LIN {X -75.070,Y -30.211,Z -61.011,A -90.000,B 90.000,C 0.000} C_DIS
LIN {X -75.157,Y -30.255,Z -61.208,A -90.000,B 90.000,C 0.000} C_DIS
LIN {X -75.236,Y -30.297,Z -61.411,A -90.000,B 90.000,C 0.000} C_DIS
LIN {X -75.317,Y -30.342,Z -61.633,A -90.000,B 90.000,C 0.000} C_DIS
LIN {X -75.352,Y -30.355,Z -61.731,A -90.000,B 90.000,C 0.000} C_DIS
LIN {X -75.467,Y -30.405,Z -62.109,A -90.000,B 90.000,C 0.000} C_DIS
LIN {X -75.521,Y -30.436,Z -62.301,A -90.000,B 90.000,C 0.000} C_DIS
LIN {X -75.551,Y -30.454,Z -62.421,A -90.000,B 90.000,C 0.000} C_DIS
LIN {X -75.584,Y -30.470,Z -62.557,A -90.000,B 90.000,C 0.000} C_DIS
LIN {X -75.622,Y -30.482,Z -62.719,A -90.000,B 90.000,C 0.000} C_DIS
LIN {X -75.673,Y -30.490,Z -62.969,A -90.000,B 90.000,C 0.000} C_DIS
LIN {X -75.693,Y -30.495,Z -63.078,A -90.000,B 90.000,C 0.000} C_DIS
LIN {X -75.763,Y -30.514,Z -63.484,A -90.000,B 90.000,C 0.000} C_DIS
LIN {X -75.780,Y -30.517,Z -63.601,A -90.000,B 90.000,C 0.000} C_DIS
LIN {X -75.801,Y -30.514,Z -63.775,A -90.000,B 90.000,C 0.000} C_DIS
LIN {X -75.817,Y -30.506,Z -63.923,A -90.000,B 90.000,C 0.000} C_DIS
LIN {X -75.841,Y -30.490,Z -64.222,A -90.000,B 90.000,C 0.000} C_DIS
LIN {X -75.855,Y -30.471,Z -64.525,A -90.000,B 90.000,C 0.000} C_DIS
LIN {X -75.859,Y -30.448,Z -64.759,A -90.000,B 90.000,C 0.000} C_DIS
LIN {X -75.857,Y -30.400,Z -65.089,A -90.000,B 90.000,C 0.000} C_DIS
LIN {X -75.852,Y -30.383,Z -65.199,A -90.000,B 90.000,C 0.000} C_DIS
LIN {X -75.840,Y -30.342,Z -65.434,A -90.000,B 90.000,C 0.000} C_DIS
LIN {X -75.824,Y -30.298,Z -65.657,A -90.000,B 90.000,C 0.000} C_DIS
LIN {X -75.790,Y -30.221,Z -66.013,A -90.000,B 90.000,C 0.000} C_DIS
LIN {X -75.781,Y -30.202,Z -66.095,A -90.000,B 90.000,C 0.000} C_DIS
LIN {X -75.717,Y -30.104,Z -66.510,A -90.000,B 90.000,C 0.000} C_DIS
LIN {X -75.684,Y -30.057,Z -66.702,A -90.000,B 90.000,C 0.000} C_DIS
LIN {X -75.646,Y -30.005,Z -66.902,A -90.000,B 90.000,C 0.000} C_DIS
LIN {X -75.556,Y -29.899,Z -67.292,A -90.000,B 90.000,C 0.000} C_DIS
LIN {X -75.456,Y -29.777,Z -67.697,A -90.000,B 90.000,C 0.000} C_DIS
LIN {X -75.421,Y -29.737,Z -67.825,A -90.000,B 90.000,C 0.000} C_DIS
LIN {X -75.365,Y -29.676,Z -68.020,A -90.000,B 90.000,C 0.000} C_DIS
LIN {X -75.295,Y -29.600,Z -68.251,A -90.000,B 90.000,C 0.000} C_DIS
LIN {X -75.175,Y -29.475,Z -68.600,A -90.000,B 90.000,C 0.000} C_DIS
LIN {X -75.139,Y -29.441,Z -68.694,A -90.000,B 90.000,C 0.000} C_DIS
LIN {X -75.103,Y -29.407,Z -68.780,A -90.000,B 90.000,C 0.000} C_DIS
LIN {X -75.036,Y -29.353,Z -68.939,A -90.000,B 90.000,C 0.000} C_DIS
LIN {X -74.986,Y -29.308,Z -69.055,A -90.000,B 90.000,C 0.000} C_DIS
LIN {X -74.986,Y -60.000,Z -69.055,A -90.000,B 90.000,C 0.000} C_DIS
LIN {X -75.487,Y -60.000,Z -57.775,A -90.000,B 90.000,C 0.000} C_DIS
LIN {X -75.487,Y -29.308,Z -57.775,A -90.000,B 90.000,C 0.000} C_DIS
LIN {X -75.588,Y -29.374,Z -57.912,A -90.000,B 90.000,C 0.000} C_DIS
LIN {X -75.705,Y -29.444,Z -58.076,A -90.000,B 90.000,C 0.000} C_DIS
LIN {X -75.899,Y -29.577,Z -58.363,A -90.000,B 90.000,C 0.000} C_DIS
LIN {X -76.016,Y -29.661,Z -58.548,A -90.000,B 90.000,C 0.000} C_DIS
LIN {X -76.226,Y -29.805,Z -58.898,A -90.000,B 90.000,C 0.000} C_DIS
LIN {X -76.268,Y -29.838,Z -58.968,A -90.000,B 90.000,C 0.000} C_DIS
LIN {X -76.317,Y -29.873,Z -59.050,A -90.000,B 90.000,C 0.000} C_DIS
LIN {X -76.378,Y -29.912,Z -59.154,A -90.000,B 90.000,C 0.000} C_DIS
LIN {X -76.468,Y -29.969,Z -59.312,A -90.000,B 90.000,C 0.000} C_DIS
LIN {X -76.540,Y -30.015,Z -59.446,A -90.000,B 90.000,C 0.000} C_DIS
LIN {X -76.686,Y -30.114,Z -59.738,A -90.000,B 90.000,C 0.000} C_DIS
LIN {X -76.865,Y -30.240,Z -60.127,A -90.000,B 90.000,C 0.000} C_DIS
LIN {X -76.997,Y -30.336,Z -60.429,A -90.000,B 90.000,C 0.000} C_DIS
LIN {X -77.105,Y -30.422,Z -60.708,A -90.000,B 90.000,C 0.000} C_DIS
LIN {X -77.183,Y -30.483,Z -60.928,A -90.000,B 90.000,C 0.000} C_DIS
LIN {X -77.250,Y -30.536,Z -61.129,A -90.000,B 90.000,C 0.000} C_DIS
LIN {X -77.333,Y -30.609,Z -61.412,A -90.000,B 90.000,C 0.000} C_DIS
LIN {X -77.363,Y -30.633,Z -61.516,A -90.000,B 90.000,C 0.000} C_DIS
LIN {X -77.423,Y -30.670,Z -61.730,A -90.000,B 90.000,C 0.000} C_DIS
LIN {X -77.467,Y -30.699,Z -61.904,A -90.000,B 90.000,C 0.000} C_DIS
LIN {X -77.546,Y -30.756,Z -62.248,A -90.000,B 90.000,C 0.000} C_DIS
LIN {X -77.612,Y -30.808,Z -62.596,A -90.000,B 90.000,C 0.000} C_DIS
LIN {X -77.629,Y -30.818,Z -62.691,A -90.000,B 90.000,C 0.000} C_DIS
LIN {X -77.639,Y -30.821,Z -62.751,A -90.000,B 90.000,C 0.000} C_DIS
LIN {X -77.695,Y -30.830,Z -63.070,A -90.000,B 90.000,C 0.000} C_DIS
LIN {X -77.728,Y -30.839,Z -63.278,A -90.000,B 90.000,C 0.000} C_DIS
LIN {X -77.744,Y -30.843,Z -63.408,A -90.000,B 90.000,C 0.000} C_DIS
LIN {X -77.759,Y -30.844,Z -63.540,A -90.000,B 90.000,C 0.000} C_DIS
LIN {X -77.780,Y -30.841,Z -63.734,A -90.000,B 90.000,C 0.000} C_DIS
LIN {X -77.808,Y -30.822,Z -64.070,A -90.000,B 90.000,C 0.000} C_DIS
LIN {X -77.823,Y -30.805,Z -64.362,A -90.000,B 90.000,C 0.000} C_DIS
LIN {X -77.830,Y -30.789,Z -64.526,A -90.000,B 90.000,C 0.000} C_DIS
LIN {X -77.835,Y -30.757,Z -64.759,A -90.000,B 90.000,C 0.000} C_DIS
LIN {X -77.834,Y -30.725,Z -64.999,A -90.000,B 90.000,C 0.000} C_DIS
LIN {X -77.832,Y -30.689,Z -65.212,A -90.000,B 90.000,C 0.000} C_DIS
LIN {X -77.815,Y -30.623,Z -65.585,A -90.000,B 90.000,C 0.000} C_DIS
LIN {X -77.791,Y -30.565,Z -65.906,A -90.000,B 90.000,C 0.000} C_DIS
LIN {X -77.756,Y -30.496,Z -66.260,A -90.000,B 90.000,C 0.000} C_DIS
LIN {X -77.732,Y -30.456,Z -66.455,A -90.000,B 90.000,C 0.000} C_DIS
LIN {X -77.659,Y -30.352,Z -66.915,A -90.000,B 90.000,C 0.000} C_DIS
LIN {X -77.634,Y -30.314,Z -67.066,A -90.000,B 90.000,C 0.000} C_DIS
LIN {X -77.579,Y -30.237,Z -67.357,A -90.000,B 90.000,C 0.000} C_DIS
LIN {X -77.481,Y -30.105,Z -67.792,A -90.000,B 90.000,C 0.000} C_DIS
LIN {X -77.383,Y -29.974,Z -68.194,A -90.000,B 90.000,C 0.000} C_DIS
LIN {X -77.376,Y -29.962,Z -68.225,A -90.000,B 90.000,C 0.000} C_DIS
LIN {X -77.320,Y -29.872,Z -68.440,A -90.000,B 90.000,C 0.000} C_DIS
LIN {X -77.199,Y -29.695,Z -68.857,A -90.000,B 90.000,C 0.000} C_DIS
LIN {X -77.135,Y -29.612,Z -69.048,A -90.000,B 90.000,C 0.000} C_DIS
LIN {X -77.071,Y -29.520,Z -69.234,A -90.000,B 90.000,C 0.000} C_DIS
LIN {X -77.025,Y -29.457,Z -69.361,A -90.000,B 90.000,C 0.000} C_DIS
LIN {X -76.963,Y -29.379,Z -69.514,A -90.000,B 90.000,C 0.000} C_DIS
LIN {X -76.909,Y -29.308,Z -69.641,A -90.000,B 90.000,C 0.000} C_DIS
LIN {X -76.877,Y -29.271,Z -69.720,A -90.000,B 90.000,C 0.000} C_DIS
LIN {X -76.826,Y -29.187,Z -69.873,A -90.000,B 90.000,C 0.000} C_DIS
LIN {X -76.806,Y -29.148,Z -69.945,A -90.000,B 90.000,C 0.000} C_DIS
LIN {X -76.778,Y -29.074,Z -70.083,A -90.000,B 90.000,C 0.000} C_DIS
LIN {X -76.770,Y -29.039,Z -70.149,A -90.000,B 90.000,C 0.000} C_DIS
LIN {X -76.764,Y -28.972,Z -70.272,A -90.000,B 90.000,C 0.000} C_DIS
LIN {X -76.772,Y -28.913,Z -70.387,A -90.000,B 90.000,C 0.000} C_DIS
LIN {X -76.792,Y -28.861,Z -70.491,A -90.000,B 90.000,C 0.000} C_DIS
LIN {X -76.824,Y -28.814,Z -70.586,A -90.000,B 90.000,C 0.000} C_DIS
LIN {X -76.844,Y -28.794,Z -70.630,A -90.000,B 90.000,C 0.000} C_DIS
LIN {X -76.892,Y -28.757,Z -70.710,A -90.000,B 90.000,C 0.000} C_DIS
LIN {X -76.950,Y -28.723,Z -70.781,A -90.000,B 90.000,C 0.000} C_DIS
LIN {X -77.017,Y -28.694,Z -70.841,A -90.000,B 90.000,C 0.000} C_DIS
LIN {X -77.054,Y -28.682,Z -70.868,A -90.000,B 90.000,C 0.000} C_DIS
LIN {X -77.132,Y -28.662,Z -70.913,A -90.000,B 90.000,C 0.000} C_DIS
LIN {X -77.218,Y -28.647,Z -70.948,A -90.000,B 90.000,C 0.000} C_DIS
LIN {X -77.310,Y -28.637,Z -70.973,A -90.000,B 90.000,C 0.000} C_DIS
LIN {X -77.406,Y -28.632,Z -70.988,A -90.000,B 90.000,C 0.000} C_DIS
LIN {X -77.456,Y -28.631,Z -70.992,A -90.000,B 90.000,C 0.000} C_DIS
LIN {X -77.559,Y -28.634,Z -70.991,A -90.000,B 90.000,C 0.000} C_DIS
LIN {X -77.612,Y -28.637,Z -70.987,A -90.000,B 90.000,C 0.000} C_DIS
LIN {X -77.719,Y -28.649,Z -70.970,A -90.000,B 90.000,C 0.000} C_DIS
LIN {X -77.774,Y -28.657,Z -70.958,A -90.000,B 90.000,C 0.000} C_DIS
LIN {X -77.884,Y -28.677,Z -70.926,A -90.000,B 90.000,C 0.000} C_DIS
LIN {X -77.994,Y -28.703,Z -70.883,A -90.000,B 90.000,C 0.000} C_DIS
LIN {X -78.104,Y -28.734,Z -70.830,A -90.000,B 90.000,C 0.000} C_DIS
LIN {X -78.159,Y -28.751,Z -70.799,A -90.000,B 90.000,C 0.000} C_DIS
LIN {X -78.267,Y -28.789,Z -70.729,A -90.000,B 90.000,C 0.000} C_DIS
LIN {X -78.373,Y -28.832,Z -70.649,A -90.000,B 90.000,C 0.000} C_DIS
LIN {X -78.425,Y -28.856,Z -70.604,A -90.000,B 90.000,C 0.000} C_DIS
LIN {X -78.525,Y -28.906,Z -70.507,A -90.000,B 90.000,C 0.000} C_DIS
LIN {X -78.622,Y -28.962,Z -70.399,A -90.000,B 90.000,C 0.000} C_DIS
LIN {X -78.713,Y -29.024,Z -70.280,A -90.000,B 90.000,C 0.000} C_DIS
LIN {X -78.798,Y -29.092,Z -70.149,A -90.000,B 90.000,C 0.000} C_DIS
LIN {X -78.877,Y -29.163,Z -70.008,A -90.000,B 90.000,C 0.000} C_DIS
LIN {X -78.947,Y -29.236,Z -69.855,A -90.000,B 90.000,C 0.000} C_DIS
LIN {X -78.979,Y -29.275,Z -69.774,A -90.000,B 90.000,C 0.000} C_DIS
LIN {X -79.009,Y -29.308,Z -69.690,A -90.000,B 90.000,C 0.000} C_DIS
LIN {X -79.097,Y -29.432,Z -69.431,A -90.000,B 90.000,C 0.000} C_DIS
LIN {X -79.136,Y -29.488,Z -69.310,A -90.000,B 90.000,C 0.000} C_DIS
LIN {X -79.250,Y -29.666,Z -68.921,A -90.000,B 90.000,C 0.000} C_DIS
LIN {X -79.335,Y -29.794,Z -68.596,A -90.000,B 90.000,C 0.000} C_DIS
LIN {X -79.365,Y -29.841,Z -68.472,A -90.000,B 90.000,C 0.000} C_DIS
LIN {X -79.464,Y -29.983,Z -68.059,A -90.000,B 90.000,C 0.000} C_DIS
LIN {X -79.538,Y -30.078,Z -67.731,A -90.000,B 90.000,C 0.000} C_DIS
LIN {X -79.614,Y -30.175,Z -67.319,A -90.000,B 90.000,C 0.000} C_DIS
LIN {X -79.633,Y -30.199,Z -67.204,A -90.000,B 90.000,C 0.000} C_DIS
LIN {X -79.716,Y -30.304,Z -66.656,A -90.000,B 90.000,C 0.000} C_DIS
LIN {X -79.743,Y -30.346,Z -66.432,A -90.000,B 90.000,C 0.000} C_DIS
LIN {X -79.782,Y -30.423,Z -66.029,A -90.000,B 90.000,C 0.000} C_DIS
LIN {X -79.809,Y -30.494,Z -65.654,A -90.000,B 90.000,C 0.000} C_DIS
LIN {X -79.829,Y -30.583,Z -65.203,A -90.000,B 90.000,C 0.000} C_DIS
LIN {X -79.832,Y -30.637,Z -64.931,A -90.000,B 90.000,C 0.000} C_DIS
LIN {X -79.831,Y -30.688,Z -64.643,A -90.000,B 90.000,C 0.000} C_DIS
LIN {X -79.826,Y -30.718,Z -64.432,A -90.000,B 90.000,C 0.000} C_DIS
LIN {X -79.812,Y -30.760,Z -64.109,A -90.000,B 90.000,C 0.000} C_DIS
LIN {X -79.800,Y -30.786,Z -63.901,A -90.000,B 90.000,C 0.000} C_DIS
LIN {X -79.776,Y -30.821,Z -63.606,A -90.000,B 90.000,C 0.000} C_DIS
LIN {X -79.748,Y -30.833,Z -63.329,A -90.000,B 90.000,C 0.000} C_DIS
LIN {X -79.709,Y -30.846,Z -63.005,A -90.000,B 90.000,C 0.000} C_DIS
LIN {X -79.682,Y -30.850,Z -62.829,A -90.000,B 90.000,C 0.000} C_DIS
LIN {X -79.652,Y -30.849,Z -62.653,A -90.000,B 90.000,C 0.000} C_DIS
LIN {X -79.597,Y -30.835,Z -62.339,A -90.000,B 90.000,C 0.000} C_DIS
LIN {X -79.527,Y -30.809,Z -61.960,A -90.000,B 90.000,C 0.000} C_DIS
LIN {X -79.497,Y -30.797,Z -61.808,A -90.000,B 90.000,C 0.000} C_DIS
LIN {X -79.476,Y -30.786,Z -61.720,A -90.000,B 90.000,C 0.000} C_DIS
LIN {X -79.404,Y -30.737,Z -61.408,A -90.000,B 90.000,C 0.000} C_DIS
LIN {X -79.348,Y -30.703,Z -61.187,A -90.000,B 90.000,C 0.000} C_DIS
LIN {X -79.256,Y -30.648,Z -60.864,A -90.000,B 90.000,C 0.000} C_DIS
LIN {X -79.165,Y -30.590,Z -60.555,A -90.000,B 90.000,C 0.000} C_DIS
LIN {X -79.089,Y -30.544,Z -60.326,A -90.000,B 90.000,C 0.000} C_DIS
LIN {X -79.019,Y -30.504,Z -60.123,A -90.000,B 90.000,C 0.000} C_DIS
LIN {X -78.959,Y -30.470,Z -59.961,A -90.000,B 90.000,C 0.000} C_DIS
LIN {X -78.853,Y -30.411,Z -59.686,A -90.000,B 90.000,C 0.000} C_DIS
LIN {X -78.755,Y -30.359,Z -59.461,A -90.000,B 90.000,C 0.000} C_DIS
LIN {X -78.672,Y -30.312,Z -59.273,A -90.000,B 90.000,C 0.000} C_DIS
LIN {X -78.596,Y -30.271,Z -59.110,A -90.000,B 90.000,C 0.000} C_DIS
LIN {X -78.494,Y -30.219,Z -58.891,A -90.000,B 90.000,C 0.000} C_DIS
LIN {X -78.326,Y -30.122,Z -58.553,A -90.000,B 90.000,C 0.000} C_DIS
LIN {X -78.288,Y -30.099,Z -58.479,A -90.000,B 90.000,C 0.000} C_DIS
LIN {X -78.218,Y -30.055,Z -58.347,A -90.000,B 90.000,C 0.000} C_DIS
LIN {X -78.075,Y -29.971,Z -58.098,A -90.000,B 90.000,C 0.000} C_DIS
LIN {X -77.857,Y -29.832,Z -57.731,A -90.000,B 90.000,C 0.000} C_DIS
LIN {X -77.697,Y -29.704,Z -57.464,A -90.000,B 90.000,C 0.000} C_DIS
LIN {X -77.595,Y -29.626,Z -57.303,A -90.000,B 90.000,C 0.000} C_DIS
LIN {X -77.526,Y -29.571,Z -57.198,A -90.000,B 90.000,C 0.000} C_DIS
LIN {X -77.371,Y -29.450,Z -56.969,A -90.000,B 90.000,C 0.000} C_DIS
LIN {X -77.219,Y -29.308,Z -56.755,A -90.000,B 90.000,C 0.000} C_DIS
LIN {X -77.219,Y -60.000,Z -56.755,A -90.000,B 90.000,C 0.000} C_DIS
LIN {X -81.350,Y -60.000,Z -68.141,A -90.000,B 90.000,C 0.000} C_DIS
LIN {X -81.350,Y -29.308,Z -68.141,A -90.000,B 90.000,C 0.000} C_DIS
LIN {X -81.402,Y -29.373,Z -67.896,A -90.000,B 90.000,C 0.000} C_DIS
LIN {X -81.465,Y -29.458,Z -67.573,A -90.000,B 90.000,C 0.000} C_DIS
LIN {X -81.521,Y -29.531,Z -67.237,A -90.000,B 90.000,C 0.000} C_DIS
LIN {X -81.592,Y -29.618,Z -66.755,A -90.000,B 90.000,C 0.000} C_DIS
LIN {X -81.618,Y -29.659,Z -66.531,A -90.000,B 90.000,C 0.000} C_DIS
LIN {X -81.648,Y -29.714,Z -66.217,A -90.000,B 90.000,C 0.000} C_DIS
LIN {X -81.663,Y -29.743,Z -66.039,A -90.000,B 90.000,C 0.000} C_DIS
LIN {X -81.678,Y -29.782,Z -65.813,A -90.000,B 90.000,C 0.000} C_DIS
LIN {X -81.694,Y -29.828,Z -65.576,A -90.000,B 90.000,C 0.000} C_DIS
LIN {X -81.701,Y -29.857,Z -65.445,A -90.000,B 90.000,C 0.000} C_DIS
LIN {X -81.721,Y -29.943,Z -65.094,A -90.000,B 90.000,C 0.000} C_DIS
LIN {X -81.731,Y -30.038,Z -64.718,A -90.000,B 90.000,C 0.000} C_DIS
LIN {X -81.733,Y -30.072,Z -64.570,A -90.000,B 90.000,C 0.000} C_DIS
LIN {X -81.733,Y -30.147,Z -64.227,A -90.000,B 90.000,C 0.000} C_DIS
LIN {X -81.724,Y -30.226,Z -63.852,A -90.000,B 90.000,C 0.000} C_DIS
LIN {X -81.716,Y -30.257,Z -63.679,A -90.000,B 90.000,C 0.000} C_DIS
LIN {X -81.701,Y -30.298,Z -63.446,A -90.000,B 90.000,C 0.000} C_DIS
LIN {X -81.674,Y -30.339,Z -63.114,A -90.000,B 90.000,C 0.000} C_DIS
LIN {X -81.627,Y -30.371,Z -62.693,A -90.000,B 90.000,C 0.000} C_DIS
LIN {X -81.593,Y -30.390,Z -62.458,A -90.000,B 90.000,C 0.000} C_DIS
LIN {X -81.549,Y -30.402,Z -62.175,A -90.000,B 90.000,C 0.000} C_DIS
LIN {X -81.528,Y -30.406,Z -62.039,A -90.000,B 90.000,C 0.000} C_DIS
LIN {X -81.477,Y -30.401,Z -61.750,A -90.000,B 90.000,C 0.000} C_DIS
LIN {X -81.442,Y -30.392,Z -61.558,A -90.000,B 90.000,C 0.000} C_DIS
LIN {X -81.416,Y -30.389,Z -61.420,A -90.000,B 90.000,C 0.000} C_DIS
LIN {X -81.399,Y -30.384,Z -61.342,A -90.000,B 90.000,C 0.000} C_DIS
LIN {X -81.384,Y -30.383,Z -61.267,A -90.000,B 90.000,C 0.000} C_DIS
LIN {X -81.312,Y -30.366,Z -60.936,A -90.000,B 90.000,C 0.000} C_DIS
LIN {X -81.256,Y -30.355,Z -60.699,A -90.000,B 90.000,C 0.000} C_DIS
LIN {X -81.162,Y -30.339,Z -60.343,A -90.000,B 90.000,C 0.000} C_DIS
LIN {X -81.080,Y -30.321,Z -60.045,A -90.000,B 90.000,C 0.000} C_DIS
LIN {X -81.050,Y -30.312,Z -59.943,A -90.000,B 90.000,C 0.000} C_DIS
LIN {X -80.964,Y -30.301,Z -59.670,A -90.000,B 90.000,C 0.000} C_DIS
LIN {X -80.864,Y -30.289,Z -59.375,A -90.000,B 90.000,C 0.000} C_DIS
LIN {X -80.828,Y -30.288,Z -59.273,A -90.000,B 90.000,C 0.000} C_DIS
LIN {X -80.786,Y -30.286,Z -59.158,A -90.000,B 90.000,C 0.000} C_DIS
LIN {X -80.714,Y -30.275,Z -58.969,A -90.000,B 90.000,C 0.000} C_DIS
LIN {X -80.639,Y -30.260,Z -58.789,A -90.000,B 90.000,C 0.000} C_DIS
LIN {X -80.544,Y -30.249,Z -58.566,A -90.000,B 90.000,C 0.000} C_DIS
LIN {X -80.414,Y -30.228,Z -58.278,A -90.000,B 90.000,C 0.000} C_DIS
LIN {X -80.309,Y -30.205,Z -58.051,A -90.000,B 90.000,C 0.000} C_DIS
LIN {X -80.245,Y -30.189,Z -57.919,A -90.000,B 90.000,C 0.000} C_DIS
LIN {X -80.160,Y -30.161,Z -57.749,A -90.000,B 90.000,C 0.000} C_DIS
LIN {X -80.048,Y -30.115,Z -57.527,A -90.000,B 90.000,C 0.000} C_DIS
LIN {X -79.993,Y -30.094,Z -57.426,A -90.000,B 90.000,C 0.000} C_DIS
LIN {X -79.803,Y -30.021,Z -57.093,A -90.000,B 90.000,C 0.000} C_DIS
LIN {X -79.744,Y -29.999,Z -56.993,A -90.000,B 90.000,C 0.000} C_DIS
LIN {X -79.506,Y -29.860,Z -56.595,A -90.000,B 90.000,C 0.000} C_DIS
LIN {X -79.371,Y -29.767,Z -56.373,A -90.000,B 90.000,C 0.000} C_DIS
LIN {X -79.307,Y -29.724,Z -56.272,A -90.000,B 90.000,C 0.000} C_DIS
LIN {X -79.170,Y -29.618,Z -56.060,A -90.000,B 90.000,C 0.000} C_DIS
LIN {X -79.030,Y -29.514,Z -55.855,A -90.000,B 90.000,C 0.000} C_DIS
LIN {X -78.810,Y -29.308,Z -55.544,A -90.000,B 90.000,C 0.000} C_DIS
LIN {X -78.614,Y -29.120,Z -55.273,A -90.000,B 90.000,C 0.000} C_DIS
LIN {X -78.524,Y -29.030,Z -55.153,A -90.000,B 90.000,C 0.000} C_DIS
LIN {X -78.438,Y -28.942,Z -55.043,A -90.000,B 90.000,C 0.000} C_DIS
LIN {X -78.357,Y -28.857,Z -54.942,A -90.000,B 90.000,C 0.000} C_DIS
LIN {X -78.281,Y -28.774,Z -54.851,A -90.000,B 90.000,C 0.000} C_DIS
LIN {X -78.210,Y -28.693,Z -54.769,A -90.000,B 90.000,C 0.000} C_DIS
LIN {X -78.143,Y -28.615,Z -54.696,A -90.000,B 90.000,C 0.000} C_DIS
LIN {X -78.081,Y -28.539,Z -54.633,A -90.000,B 90.000,C 0.000} C_DIS
LIN {X -77.970,Y -28.403,Z -54.532,A -90.000,B 90.000,C 0.000} C_DIS
LIN {X -77.921,Y -28.357,Z -54.494,A -90.000,B 90.000,C 0.000} C_DIS
LIN {X -77.876,Y -28.317,Z -54.465,A -90.000,B 90.000,C 0.000} C_DIS
LIN {X -77.835,Y -28.283,Z -54.444,A -90.000,B 90.000,C 0.000} C_DIS
LIN {X -77.782,Y -28.246,Z -54.427,A -90.000,B 90.000,C 0.000} C_DIS
LIN {X -77.752,Y -28.230,Z -54.426,A -90.000,B 90.000,C 0.000} C_DIS
LIN {X -77.738,Y -28.225,Z -54.428,A -90.000,B 90.000,C 0.000} C_DIS
LIN {X -77.714,Y -28.220,Z -54.438,A -90.000,B 90.000,C 0.000} C_DIS
LIN {X -77.693,Y -28.223,Z -54.455,A -90.000,B 90.000,C 0.000} C_DIS
LIN {X -77.684,Y -28.227,Z -54.467,A -90.000,B 90.000,C 0.000} C_DIS
LIN {X -77.670,Y -28.241,Z -54.495,A -90.000,B 90.000,C 0.000} C_DIS
LIN {X -77.658,Y -28.261,Z -54.530,A -90.000,B 90.000,C 0.000} C_DIS
LIN {X -77.648,Y -28.303,Z -54.595,A -90.000,B 90.000,C 0.000} C_DIS
LIN {X -77.646,Y -28.337,Z -54.646,A -90.000,B 90.000,C 0.000} C_DIS
LIN {X -77.652,Y -28.421,Z -54.768,A -90.000,B 90.000,C 0.000} C_DIS
LIN {X -77.660,Y -28.469,Z -54.838,A -90.000,B 90.000,C 0.000} C_DIS
LIN {X -77.685,Y -28.577,Z -54.995,A -90.000,B 90.000,C 0.000} C_DIS
LIN {X -77.747,Y -28.769,Z -55.271,A -90.000,B 90.000,C 0.000} C_DIS
LIN {X -77.802,Y -28.916,Z -55.480,A -90.000,B 90.000,C 0.000} C_DIS
LIN {X -77.834,Y -28.990,Z -55.592,A -90.000,B 90.000,C 0.000} C_DIS
LIN {X -77.906,Y -29.137,Z -55.829,A -90.000,B 90.000,C 0.000} C_DIS
LIN {X -77.946,Y -29.208,Z -55.953,A -90.000,B 90.000,C 0.000} C_DIS
LIN {X -77.988,Y -29.278,Z -56.082,A -90.000,B 90.000,C 0.000} C_DIS
LIN {X -78.033,Y -29.346,Z -56.214,A -90.000,B 90.000,C 0.000} C_DIS
LIN {X -78.080,Y -29.411,Z -56.350,A -90.000,B 90.000,C 0.000} C_DIS
LIN {X -78.129,Y -29.486,Z -56.490,A -90.000,B 90.000,C 0.000} C_DIS
LIN {X -78.235,Y -29.629,Z -56.778,A -90.000,B 90.000,C 0.000} C_DIS
LIN {X -78.348,Y -29.756,Z -57.079,A -90.000,B 90.000,C 0.000} C_DIS
LIN {X -78.470,Y -29.868,Z -57.390,A -90.000,B 90.000,C 0.000} C_DIS
LIN {X -78.598,Y -29.981,Z -57.710,A -90.000,B 90.000,C 0.000} C_DIS
LIN {X -78.734,Y -30.079,Z -58.037,A -90.000,B 90.000,C 0.000} C_DIS
LIN {X -78.875,Y -30.163,Z -58.371,A -90.000,B 90.000,C 0.000} C_DIS
LIN {X -79.022,Y -30.244,Z -58.711,A -90.000,B 90.000,C 0.000} C_DIS
LIN {X -79.174,Y -30.317,Z -59.053,A -90.000,B 90.000,C 0.000} C_DIS
LIN {X -79.330,Y -30.377,Z -59.399,A -90.000,B 90.000,C 0.000} C_DIS
LIN {X -79.490,Y -30.440,Z -59.745,A -90.000,B 90.000,C 0.000} C_DIS
LIN {X -79.654,Y -30.500,Z -60.091,A -90.000,B 90.000,C 0.000} C_DIS
LIN {X -79.820,Y -30.551,Z -60.435,A -90.000,B 90.000,C 0.000} C_DIS
LIN {X -79.989,Y -30.596,Z -60.776,A -90.000,B 90.000,C 0.000} C_DIS
LIN {X -80.159,Y -30.632,Z -61.113,A -90.000,B 90.000,C 0.000} C_DIS
LIN {X -80.331,Y -30.651,Z -61.443,A -90.000,B 90.000,C 0.000} C_DIS
LIN {X -80.503,Y -30.664,Z -61.767,A -90.000,B 90.000,C 0.000} C_DIS
LIN {X -80.589,Y -30.663,Z -61.926,A -90.000,B 90.000,C 0.000} C_DIS
LIN {X -80.675,Y -30.656,Z -62.083,A -90.000,B 90.000,C 0.000} C_DIS
LIN {X -80.761,Y -30.642,Z -62.237,A -90.000,B 90.000,C 0.000} C_DIS
LIN {X -81.018,Y -30.587,Z -62.683,A -90.000,B 90.000,C 0.000} C_DIS
LIN {X -81.103,Y -30.565,Z -62.826,A -90.000,B 90.000,C 0.000} C_DIS
LIN {X -81.187,Y -30.537,Z -62.965,A -90.000,B 90.000,C 0.000} C_DIS
LIN {X -81.271,Y -30.504,Z -63.101,A -90.000,B 90.000,C 0.000} C_DIS
LIN {X -81.354,Y -30.465,Z -63.233,A -90.000,B 90.000,C 0.000} C_DIS
LIN {X -81.437,Y -30.420,Z -63.362,A -90.000,B 90.000,C 0.000} C_DIS
LIN {X -81.518,Y -30.372,Z -63.486,A -90.000,B 90.000,C 0.000} C_DIS
LIN {X -81.599,Y -30.322,Z -63.606,A -90.000,B 90.000,C 0.000} C_DIS
LIN {X -81.680,Y -30.269,Z -63.722,A -90.000,B 90.000,C 0.000} C_DIS
LIN {X -81.759,Y -30.215,Z -63.834,A -90.000,B 90.000,C 0.000} C_DIS
LIN {X -81.914,Y -30.104,Z -64.043,A -90.000,B 90.000,C 0.000} C_DIS
LIN {X -81.990,Y -30.047,Z -64.140,A -90.000,B 90.000,C 0.000} C_DIS
LIN {X -82.064,Y -29.988,Z -64.232,A -90.000,B 90.000,C 0.000} C_DIS
LIN {X -82.138,Y -29.927,Z -64.319,A -90.000,B 90.000,C 0.000} C_DIS
LIN {X -82.210,Y -29.866,Z -64.400,A -90.000,B 90.000,C 0.000} C_DIS
LIN {X -82.281,Y -29.804,Z -64.476,A -90.000,B 90.000,C 0.000} C_DIS
LIN {X -82.350,Y -29.742,Z -64.545,A -90.000,B 90.000,C 0.000} C_DIS
LIN {X -82.417,Y -29.680,Z -64.609,A -90.000,B 90.000,C 0.000} C_DIS
LIN {X -82.483,Y -29.618,Z -64.667,A -90.000,B 90.000,C 0.000} C_DIS
LIN {X -82.547,Y -29.557,Z -64.718,A -90.000,B 90.000,C 0.000} C_DIS
LIN {X -82.640,Y -29.468,Z -64.783,A -90.000,B 90.000,C 0.000} C_DIS
LIN {X -82.729,Y -29.381,Z -64.832,A -90.000,B 90.000,C 0.000} C_DIS
LIN {X -82.813,Y -29.299,Z -64.866,A -90.000,B 90.000,C 0.000} C_DIS
LIN {X -82.893,Y -29.225,Z -64.883,A -90.000,B 90.000,C 0.000} C_DIS
LIN {X -82.968,Y -29.161,Z -64.884,A -90.000,B 90.000,C 0.000} C_DIS
LIN {X -83.015,Y -29.125,Z -64.874,A -90.000,B 90.000,C 0.000} C_DIS
LIN {X -83.037,Y -29.108,Z -64.867,A -90.000,B 90.000,C 0.000} C_DIS
LIN {X -83.081,Y -29.079,Z -64.845,A -90.000,B 90.000,C 0.000} C_DIS
LIN {X -83.122,Y -29.055,Z -64.816,A -90.000,B 90.000,C 0.000} C_DIS
LIN {X -83.141,Y -29.044,Z -64.798,A -90.000,B 90.000,C 0.000} C_DIS
LIN {X -83.178,Y -29.027,Z -64.756,A -90.000,B 90.000,C 0.000} C_DIS
LIN {X -83.213,Y -29.015,Z -64.705,A -90.000,B 90.000,C 0.000} C_DIS
LIN {X -83.245,Y -29.008,Z -64.646,A -90.000,B 90.000,C 0.000} C_DIS
LIN {X -83.274,Y -29.008,Z -64.578,A -90.000,B 90.000,C 0.000} C_DIS
LIN {X -83.300,Y -29.013,Z -64.500,A -90.000,B 90.000,C 0.000} C_DIS
LIN {X -83.323,Y -29.023,Z -64.413,A -90.000,B 90.000,C 0.000} C_DIS
LIN {X -83.344,Y -29.037,Z -64.317,A -90.000,B 90.000,C 0.000} C_DIS
LIN {X -83.361,Y -29.053,Z -64.211,A -90.000,B 90.000,C 0.000} C_DIS
LIN {X -83.375,Y -29.075,Z -64.096,A -90.000,B 90.000,C 0.000} C_DIS
LIN {X -83.390,Y -29.117,Z -63.903,A -90.000,B 90.000,C 0.000} C_DIS
LIN {X -83.396,Y -29.151,Z -63.763,A -90.000,B 90.000,C 0.000} C_DIS
LIN {X -83.399,Y -29.184,Z -63.611,A -90.000,B 90.000,C 0.000} C_DIS
LIN {X -83.399,Y -29.215,Z -63.450,A -90.000,B 90.000,C 0.000} C_DIS
LIN {X -83.387,Y -29.280,Z -63.094,A -90.000,B 90.000,C 0.000} C_DIS
LIN {X -83.375,Y -29.308,Z -62.899,A -90.000,B 90.000,C 0.000} C_DIS
LIN {X -83.340,Y -29.392,Z -62.367,A -90.000,B 90.000,C 0.000} C_DIS
LIN {X -83.321,Y -29.434,Z -62.141,A -90.000,B 90.000,C 0.000} C_DIS
LIN {X -83.293,Y -29.471,Z -61.871,A -90.000,B 90.000,C 0.000} C_DIS
LIN {X -83.279,Y -29.487,Z -61.740,A -90.000,B 90.000,C 0.000} C_DIS
LIN {X -83.251,Y -29.525,Z -61.458,A -90.000,B 90.000,C 0.000} C_DIS
LIN {X -83.233,Y -29.543,Z -61.294,A -90.000,B 90.000,C 0.000} C_DIS
LIN {X -83.206,Y -29.576,Z -61.053,A -90.000,B 90.000,C 0.000} C_DIS
LIN {X -83.177,Y -29.602,Z -60.844,A -90.000,B 90.000,C 0.000} C_DIS
LIN {X -83.140,Y -29.653,Z -60.548,A -90.000,B 90.000,C 0.000} C_DIS
LIN {X -83.085,Y -29.698,Z -60.228,A -90.000,B 90.000,C 0.000} C_DIS
LIN {X -83.039,Y -29.734,Z -59.992,A -90.000,B 90.000,C 0.000} C_DIS
LIN {X -83.018,Y -29.753,Z -59.880,A -90.000,B 90.000,C 0.000} C_DIS
LIN {X -82.978,Y -29.784,Z -59.689,A -90.000,B 90.000,C 0.000} C_DIS
LIN {X -82.952,Y -29.805,Z -59.564,A -90.000,B 90.000,C 0.000} C_DIS
LIN {X -82.909,Y -29.828,Z -59.388,A -90.000,B 90.000,C 0.000} C_DIS
LIN {X -82.831,Y -29.867,Z -59.101,A -90.000,B 90.000,C 0.000} C_DIS
LIN {X -82.800,Y -29.883,Z -58.994,A -90.000,B 90.000,C 0.000} C_DIS
LIN {X -82.745,Y -29.914,Z -58.807,A -90.000,B 90.000,C 0.000} C_DIS
LIN {X -82.687,Y -29.932,Z -58.625,A -90.000,B 90.000,C 0.000} C_DIS
LIN {X -82.667,Y -29.935,Z -58.567,A -90.000,B 90.000,C 0.000} C_DIS
LIN {X -82.629,Y -29.950,Z -58.459,A -90.000,B 90.000,C 0.000} C_DIS
LIN {X -82.569,Y -29.967,Z -58.287,A -90.000,B 90.000,C 0.000} C_DIS
LIN {X -82.465,Y -29.987,Z -58.020,A -90.000,B 90.000,C 0.000} C_DIS
LIN {X -82.412,Y -29.996,Z -57.890,A -90.000,B 90.000,C 0.000} C_DIS
LIN {X -82.280,Y -30.022,Z -57.579,A -90.000,B 90.000,C 0.000} C_DIS
LIN {X -82.107,Y -30.032,Z -57.192,A -90.000,B 90.000,C 0.000} C_DIS
LIN {X -81.997,Y -30.031,Z -56.962,A -90.000,B 90.000,C 0.000} C_DIS
LIN {X -81.911,Y -30.024,Z -56.787,A -90.000,B 90.000,C 0.000} C_DIS
LIN {X -81.809,Y -30.011,Z -56.586,A -90.000,B 90.000,C 0.000} C_DIS
LIN {X -81.720,Y -29.990,Z -56.422,A -90.000,B 90.000,C 0.000} C_DIS
LIN {X -81.578,Y -29.953,Z -56.170,A -90.000,B 90.000,C 0.000} C_DIS
LIN {X -81.449,Y -29.911,Z -55.951,A -90.000,B 90.000,C 0.000} C_DIS
LIN {X -81.328,Y -29.870,Z -55.746,A -90.000,B 90.000,C 0.000} C_DIS
LIN {X -81.274,Y -29.847,Z -55.655,A -90.000,B 90.000,C 0.000} C_DIS
LIN {X -81.057,Y -29.725,Z -55.297,A -90.000,B 90.000,C 0.000} C_DIS
LIN {X -81.027,Y -29.707,Z -55.250,A -90.000,B 90.000,C 0.000} C_DIS
LIN {X -80.840,Y -29.582,Z -54.961,A -90.000,B 90.000,C 0.000} C_DIS
LIN {X -80.659,Y -29.453,Z -54.695,A -90.000,B 90.000,C 0.000} C_DIS
LIN {X -80.550,Y -29.376,Z -54.540,A -90.000,B 90.000,C 0.000} C_DIS
LIN {X -80.478,Y -29.308,Z -54.439,A -90.000,B 90.000,C 0.000} C_DIS
LIN {X -80.342,Y -29.188,Z -54.248,A -90.000,B 90.000,C 0.000} C_DIS
LIN {X -80.223,Y -29.065,Z -54.084,A -90.000,B 90.000,C 0.000} C_DIS
LIN {X -80.032,Y -28.856,Z -53.832,A -90.000,B 90.000,C 0.000} C_DIS
LIN {X -79.960,Y -28.781,Z -53.742,A -90.000,B 90.000,C 0.000} C_DIS
LIN {X -79.879,Y -28.699,Z -53.651,A -90.000,B 90.000,C 0.000} C_DIS
LIN {X -79.843,Y -28.665,Z -53.617,A -90.000,B 90.000,C 0.000} C_DIS
LIN {X -79.830,Y -28.655,Z -53.608,A -90.000,B 90.000,C 0.000} C_DIS
LIN {X -79.820,Y -28.648,Z -53.604,A -90.000,B 90.000,C 0.000} C_DIS
LIN {X -79.814,Y -28.647,Z -53.605,A -90.000,B 90.000,C 0.000} C_DIS
LIN {X -79.810,Y -28.649,Z -53.611,A -90.000,B 90.000,C 0.000} C_DIS
LIN {X -79.810,Y -28.656,Z -53.622,A -90.000,B 90.000,C 0.000} C_DIS
LIN {X -79.819,Y -28.681,Z -53.657,A -90.000,B 90.000,C 0.000} C_DIS
LIN {X -79.871,Y -28.773,Z -53.780,A -90.000,B 90.000,C 0.000} C_DIS
LIN {X -79.966,Y -28.911,Z -53.966,A -90.000,B 90.000,C 0.000} C_DIS
LIN {X -80.100,Y -29.094,Z -54.208,A -90.000,B 90.000,C 0.000} C_DIS
LIN {X -80.181,Y -29.193,Z -54.348,A -90.000,B 90.000,C 0.000} C_DIS
LIN {X -80.270,Y -29.292,Z -54.500,A -90.000,B 90.000,C 0.000} C_DIS
LIN {X -80.366,Y -29.388,Z -54.662,A -90.000,B 90.000,C 0.000} C_DIS
LIN {X -80.470,Y -29.479,Z -54.834,A -90.000,B 90.000,C 0.000} C_DIS
LIN {X -80.580,Y -29.564,Z -55.015,A -90.000,B 90.000,C 0.000} C_DIS
LIN {X -80.819,Y -29.730,Z -55.399,A -90.000,B 90.000,C 0.000} C_DIS
LIN {X -80.947,Y -29.806,Z -55.601,A -90.000,B 90.000,C 0.000} C_DIS
LIN {X -81.080,Y -29.871,Z -55.808,A -90.000,B 90.000,C 0.000} C_DIS
LIN {X -81.216,Y -29.924,Z -56.020,A -90.000,B 90.000,C 0.000} C_DIS
LIN {X -81.357,Y -29.963,Z -56.234,A -90.000,B 90.000,C 0.000} C_DIS
LIN {X -81.501,Y -29.996,Z -56.452,A -90.000,B 90.000,C 0.000} C_DIS
LIN {X -81.648,Y -30.026,Z -56.671,A -90.000,B 90.000,C 0.000} C_DIS
LIN {X -81.797,Y -30.043,Z -56.891,A -90.000,B 90.000,C 0.000} C_DIS
LIN {X -81.947,Y -30.046,Z -57.110,A -90.000,B 90.000,C 0.000} C_DIS
LIN {X -82.252,Y -30.026,Z -57.546,A -90.000,B 90.000,C 0.000} C_DIS
LIN {X -82.405,Y -30.002,Z -57.760,A -90.000,B 90.000,C 0.000} C_DIS
LIN {X -82.558,Y -29.976,Z -57.971,A -90.000,B 90.000,C 0.000} C_DIS
LIN {X -82.710,Y -29.944,Z -58.176,A -90.000,B 90.000,C 0.000} C_DIS
LIN {X -83.011,Y -29.858,Z -58.571,A -90.000,B 90.000,C 0.000} C_DIS
LIN {X -83.158,Y -29.805,Z -58.758,A -90.000,B 90.000,C 0.000} C_DIS
LIN {X -83.302,Y -29.748,Z -58.937,A -90.000,B 90.000,C 0.000} C_DIS
LIN {X -83.443,Y -29.691,Z -59.106,A -90.000,B 90.000,C 0.000} C_DIS
LIN {X -83.581,Y -29.625,Z -59.266,A -90.000,B 90.000,C 0.000} C_DIS
LIN {X -83.714,Y -29.558,Z -59.415,A -90.000,B 90.000,C 0.000} C_DIS
LIN {X -83.843,Y -29.493,Z -59.553,A -90.000,B 90.000,C 0.000} C_DIS
LIN {X -83.967,Y -29.425,Z -59.678,A -90.000,B 90.000,C 0.000} C_DIS
LIN {X -84.026,Y -29.390,Z -59.735,A -90.000,B 90.000,C 0.000} C_DIS
LIN {X -84.196,Y -29.288,Z -59.886,A -90.000,B 90.000,C 0.000} C_DIS
LIN {X -84.301,Y -29.227,Z -59.968,A -90.000,B 90.000,C 0.000} C_DIS
LIN {X -84.399,Y -29.170,Z -60.034,A -90.000,B 90.000,C 0.000} C_DIS
LIN {X -84.445,Y -29.142,Z -60.060,A -90.000,B 90.000,C 0.000} C_DIS
LIN {X -84.531,Y -29.092,Z -60.100,A -90.000,B 90.000,C 0.000} C_DIS
LIN {X -84.571,Y -29.070,Z -60.113,A -90.000,B 90.000,C 0.000} C_DIS
LIN {X -84.609,Y -29.050,Z -60.122,A -90.000,B 90.000,C 0.000} C_DIS
LIN {X -84.644,Y -29.032,Z -60.125,A -90.000,B 90.000,C 0.000} C_DIS
LIN {X -84.693,Y -29.010,Z -60.122,A -90.000,B 90.000,C 0.000} C_DIS
LIN {X -84.723,Y -28.999,Z -60.113,A -90.000,B 90.000,C 0.000} C_DIS
LIN {X -84.763,Y -28.988,Z -60.090,A -90.000,B 90.000,C 0.000} C_DIS
LIN {X -84.787,Y -28.984,Z -60.068,A -90.000,B 90.000,C 0.000} C_DIS
LIN {X -84.817,Y -28.983,Z -60.024,A -90.000,B 90.000,C 0.000} C_DIS
LIN {X -84.834,Y -28.987,Z -59.988,A -90.000,B 90.000,C 0.000} C_DIS
LIN {X -84.854,Y -28.998,Z -59.924,A -90.000,B 90.000,C 0.000} C_DIS
LIN {X -84.864,Y -29.009,Z -59.873,A -90.000,B 90.000,C 0.000} C_DIS
LIN {X -84.875,Y -29.040,Z -59.754,A -90.000,B 90.000,C 0.000} C_DIS
LIN {X -84.874,Y -29.080,Z -59.609,A -90.000,B 90.000,C 0.000} C_DIS
LIN {X -84.860,Y -29.128,Z -59.439,A -90.000,B 90.000,C 0.000} C_DIS
LIN {X -84.833,Y -29.182,Z -59.242,A -90.000,B 90.000,C 0.000} C_DIS
LIN {X -84.792,Y -29.246,Z -59.018,A -90.000,B 90.000,C 0.000} C_DIS
LIN {X -84.767,Y -29.281,Z -58.895,A -90.000,B 90.000,C 0.000} C_DIS
LIN {X -84.738,Y -29.308,Z -58.764,A -90.000,B 90.000,C 0.000} C_DIS
LIN {X -84.700,Y -29.353,Z -58.602,A -90.000,B 90.000,C 0.000} C_DIS
LIN {X -84.641,Y -29.410,Z -58.370,A -90.000,B 90.000,C 0.000} C_DIS
LIN {X -84.614,Y -29.435,Z -58.271,A -90.000,B 90.000,C 0.000} C_DIS
LIN {X -84.542,Y -29.484,Z -58.027,A -90.000,B 90.000,C 0.000} C_DIS
LIN {X -84.492,Y -29.517,Z -57.865,A -90.000,B 90.000,C 0.000} C_DIS
LIN {X -84.412,Y -29.565,Z -57.622,A -90.000,B 90.000,C 0.000} C_DIS
LIN {X -84.377,Y -29.588,Z -57.520,A -90.000,B 90.000,C 0.000} C_DIS
LIN {X -84.248,Y -29.648,Z -57.176,A -90.000,B 90.000,C 0.000} C_DIS
LIN {X -84.198,Y -29.670,Z -57.049,A -90.000,B 90.000,C 0.000} C_DIS
LIN {X -84.050,Y -29.714,Z -56.695,A -90.000,B 90.000,C 0.000} C_DIS
LIN {X -83.892,Y -29.751,Z -56.334,A -90.000,B 90.000,C 0.000} C_DIS
LIN {X -83.785,Y -29.772,Z -56.104,A -90.000,B 90.000,C 0.000} C_DIS
LIN {X -83.688,Y -29.788,Z -55.901,A -90.000,B 90.000,C 0.000} C_DIS
LIN {X -83.607,Y -29.794,Z -55.737,A -90.000,B 90.000,C 0.000} C_DIS
LIN {X -83.523,Y -29.792,Z -55.574,A -90.000,B 90.000,C 0.000} C_DIS
LIN {X -83.447,Y -29.786,Z -55.433,A -90.000,B 90.000,C 0.000} C_DIS
LIN {X -83.312,Y -29.763,Z -55.191,A -90.000,B 90.000,C 0.000} C_DIS
LIN {X -83.183,Y -29.739,Z -54.968,A -90.000,B 90.000,C 0.000} C_DIS
LIN {X -83.018,Y -29.694,Z -54.688,A -90.000,B 90.000,C 0.000} C_DIS
LIN {X -82.898,Y -29.656,Z -54.486,A -90.000,B 90.000,C 0.000} C_DIS
LIN {X -82.869,Y -29.645,Z -54.437,A -90.000,B 90.000,C 0.000} C_DIS
LIN {X -82.723,Y -29.568,Z -54.198,A -90.000,B 90.000,C 0.000} C_DIS
LIN {X -82.623,Y -29.517,Z -54.043,A -90.000,B 90.000,C 0.000} C_DIS
LIN {X -82.518,Y -29.450,Z -53.880,A -90.000,B 90.000,C 0.000} C_DIS
LIN {X -82.351,Y -29.343,Z -53.634,A -90.000,B 90.000,C 0.000} C_DIS
LIN {X -82.301,Y -29.308,Z -53.563,A -90.000,B 90.000,C 0.000} C_DIS
LIN {X -82.104,Y -29.167,Z -53.273,A -90.000,B 90.000,C 0.000} C_DIS
LIN {X -82.026,Y -29.099,Z -53.157,A -90.000,B 90.000,C 0.000} C_DIS
LIN {X -81.963,Y -29.037,Z -53.059,A -90.000,B 90.000,C 0.000} C_DIS
LIN {X -81.874,Y -28.941,Z -52.917,A -90.000,B 90.000,C 0.000} C_DIS
LIN {X -81.841,Y -28.897,Z -52.854,A -90.000,B 90.000,C 0.000} C_DIS
LIN {X -81.833,Y -28.883,Z -52.832,A -90.000,B 90.000,C 0.000} C_DIS
LIN {X -81.834,Y -28.879,Z -52.825,A -90.000,B 90.000,C 0.000} C_DIS
LIN {X -81.850,Y -28.887,Z -52.831,A -90.000,B 90.000,C 0.000} C_DIS
LIN {X -81.890,Y -28.917,Z -52.866,A -90.000,B 90.000,C 0.000} C_DIS
LIN {X -81.977,Y -28.987,Z -52.957,A -90.000,B 90.000,C 0.000} C_DIS
LIN {X -82.099,Y -29.081,Z -53.092,A -90.000,B 90.000,C 0.000} C_DIS
LIN {X -82.251,Y -29.188,Z -53.268,A -90.000,B 90.000,C 0.000} C_DIS
LIN {X -82.432,Y -29.297,Z -53.478,A -90.000,B 90.000,C 0.000} C_DIS
LIN {X -82.636,Y -29.404,Z -53.717,A -90.000,B 90.000,C 0.000} C_DIS
LIN {X -82.860,Y -29.515,Z -53.981,A -90.000,B 90.000,C 0.000} C_DIS
LIN {X -83.101,Y -29.604,Z -54.264,A -90.000,B 90.000,C 0.000} C_DIS
LIN {X -83.355,Y -29.665,Z -54.560,A -90.000,B 90.000,C 0.000} C_DIS
LIN {X -83.618,Y -29.696,Z -54.865,A -90.000,B 90.000,C 0.000} C_DIS
LIN {X -83.887,Y -29.716,Z -55.173,A -90.000,B 90.000,C 0.000} C_DIS
LIN {X -84.158,Y -29.703,Z -55.479,A -90.000,B 90.000,C 0.000} C_DIS
LIN {X -84.293,Y -29.684,Z -55.629,A -90.000,B 90.000,C 0.000} C_DIS
LIN {X -84.427,Y -29.662,Z -55.778,A -90.000,B 90.000,C 0.000} C_DIS
LIN {X -84.560,Y -29.638,Z -55.923,A -90.000,B 90.000,C 0.000} C_DIS
LIN {X -84.691,Y -29.609,Z -56.064,A -90.000,B 90.000,C 0.000} C_DIS
LIN {X -84.947,Y -29.547,Z -56.333,A -90.000,B 90.000,C 0.000} C_DIS
LIN {X -85.070,Y -29.512,Z -56.459,A -90.000,B 90.000,C 0.000} C_DIS
LIN {X -85.306,Y -29.440,Z -56.691,A -90.000,B 90.000,C 0.000} C_DIS
LIN {X -85.417,Y -29.404,Z -56.796,A -90.000,B 90.000,C 0.000} C_DIS
LIN {X -85.624,Y -29.329,Z -56.980,A -90.000,B 90.000,C 0.000} C_DIS
LIN {X -85.719,Y -29.296,Z -57.058,A -90.000,B 90.000,C 0.000} C_DIS
LIN {X -85.850,Y -29.249,Z -57.156,A -90.000,B 90.000,C 0.000} C_DIS
LIN {X -85.965,Y -29.205,Z -57.228,A -90.000,B 90.000,C 0.000} C_DIS
LIN {X -86.033,Y -29.179,Z -57.261,A -90.000,B 90.000,C 0.000} C_DIS
LIN {X -86.063,Y -29.169,Z -57.272,A -90.000,B 90.000,C 0.000} C_DIS
LIN {X -86.118,Y -29.151,Z -57.286,A -90.000,B 90.000,C 0.000} C_DIS
LIN {X -86.142,Y -29.144,Z -57.287,A -90.000,B 90.000,C 0.000} C_DIS
LIN {X -86.174,Y -29.136,Z -57.283,A -90.000,B 90.000,C 0.000} C_DIS
LIN {X -86.193,Y -29.132,Z -57.275,A -90.000,B 90.000,C 0.000} C_DIS
LIN {X -86.209,Y -29.129,Z -57.264,A -90.000,B 90.000,C 0.000} C_DIS
LIN {X -86.229,Y -29.127,Z -57.239,A -90.000,B 90.000,C 0.000} C_DIS
LIN {X -86.239,Y -29.128,Z -57.218,A -90.000,B 90.000,C 0.000} C_DIS
LIN {X -86.251,Y -29.133,Z -57.164,A -90.000,B 90.000,C 0.000} C_DIS
LIN {X -86.252,Y -29.144,Z -57.093,A -90.000,B 90.000,C 0.000} C_DIS
LIN {X -86.242,Y -29.160,Z -57.004,A -90.000,B 90.000,C 0.000} C_DIS
LIN {X -86.220,Y -29.183,Z -56.897,A -90.000,B 90.000,C 0.000} C_DIS
LIN {X -86.186,Y -29.210,Z -56.771,A -90.000,B 90.000,C 0.000} C_DIS
LIN {X -86.111,Y -29.256,Z -56.546,A -90.000,B 90.000,C 0.000} C_DIS
LIN {X -86.006,Y -29.308,Z -56.275,A -90.000,B 90.000,C 0.000} C_DIS
LIN {X -85.924,Y -29.344,Z -56.073,A -90.000,B 90.000,C 0.000} C_DIS
LIN {X -85.808,Y -29.390,Z -55.796,A -90.000,B 90.000,C 0.000} C_DIS
LIN {X -85.662,Y -29.428,Z -55.461,A -90.000,B 90.000,C 0.000} C_DIS
LIN {X -85.570,Y -29.450,Z -55.262,A -90.000,B 90.000,C 0.000} C_DIS
LIN {X -85.431,Y -29.480,Z -54.968,A -90.000,B 90.000,C 0.000} C_DIS
LIN {X -85.268,Y -29.500,Z -54.643,A -90.000,B 90.000,C 0.000} C_DIS
LIN {X -85.190,Y -29.506,Z -54.493,A -90.000,B 90.000,C 0.000} C_DIS
LIN {X -85.104,Y -29.506,Z -54.336,A -90.000,B 90.000,C 0.000} C_DIS
LIN {X -85.019,Y -29.498,Z -54.182,A -90.000,B 90.000,C 0.000} C_DIS
LIN {X -84.925,Y -29.483,Z -54.019,A -90.000,B 90.000,C 0.000} C_DIS
LIN {X -84.752,Y -29.446,Z -53.723,A -90.000,B 90.000,C 0.000} C_DIS
LIN {X -84.519,Y -29.382,Z -53.327,A -90.000,B 90.000,C 0.000} C_DIS
LIN {X -84.442,Y -29.353,Z -53.199,A -90.000,B 90.000,C 0.000} C_DIS
LIN {X -84.354,Y -29.308,Z -53.061,A -90.000,B 90.000,C 0.000} C_DIS
LIN {X -84.354,Y -60.000,Z -53.061,A -90.000,B 90.000,C 0.000} C_DIS
LIN {X -0.780,Y -60.000,Z -174.323,A -90.000,B 90.000,C 0.000} C_DIS
LIN {X -0.780,Y -29.308,Z -174.323,A -90.000,B 90.000,C 0.000} C_DIS
LIN {X 0.285,Y -29.408,Z -172.922,A -90.000,B 90.000,C 0.000} C_DIS
LIN {X 0.476,Y -29.432,Z -172.664,A -90.000,B 90.000,C 0.000} C_DIS
LIN {X 0.526,Y -29.437,Z -172.592,A -90.000,B 90.000,C 0.000} C_DIS
LIN {X 1.168,Y -29.528,Z -171.619,A -90.000,B 90.000,C 0.000} C_DIS
LIN {X 1.225,Y -29.534,Z -171.527,A -90.000,B 90.000,C 0.000} C_DIS
LIN {X 1.303,Y -29.539,Z -171.382,A -90.000,B 90.000,C 0.000} C_DIS
LIN {X 1.611,Y -29.578,Z -170.796,A -90.000,B 90.000,C 0.000} C_DIS
LIN {X 2.222,Y -29.661,Z -169.666,A -90.000,B 90.000,C 0.000} C_DIS
LIN {X 2.395,Y -29.675,Z -169.288,A -90.000,B 90.000,C 0.000} C_DIS
LIN {X 2.446,Y -29.675,Z -169.155,A -90.000,B 90.000,C 0.000} C_DIS
LIN {X 2.484,Y -29.682,Z -169.048,A -90.000,B 90.000,C 0.000} C_DIS
LIN {X 2.596,Y -29.707,Z -168.728,A -90.000,B 90.000,C 0.000} C_DIS
LIN {X 2.648,Y -29.716,Z -168.527,A -90.000,B 90.000,C 0.000} C_DIS
LIN {X 2.779,Y -29.724,Z -168.058,A -90.000,B 90.000,C 0.000} C_DIS
LIN {X 3.008,Y -29.742,Z -167.256,A -90.000,B 90.000,C 0.000} C_DIS
LIN {X 3.099,Y -29.731,Z -166.793,A -90.000,B 90.000,C 0.000} C_DIS
LIN {X 3.117,Y -29.732,Z -166.697,A -90.000,B 90.000,C 0.000} C_DIS
LIN {X 3.127,Y -29.729,Z -166.595,A -90.000,B 90.000,C 0.000} C_DIS
LIN {X 3.129,Y -29.712,Z -166.346,A -90.000,B 90.000,C 0.000} C_DIS
LIN {X 3.152,Y -29.677,Z -165.711,A -90.000,B 90.000,C 0.000} C_DIS
LIN {X 3.157,Y -29.684,Z -165.370,A -90.000,B 90.000,C 0.000} C_DIS
LIN {X 3.166,Y -29.691,Z -165.145,A -90.000,B 90.000,C 0.000} C_DIS
LIN {X 3.169,Y -29.700,Z -165.032,A -90.000,B 90.000,C 0.000} C_DIS
LIN {X 3.051,Y -29.699,Z -164.287,A -90.000,B 90.000,C 0.000} C_DIS
LIN {X 2.909,Y -29.653,Z -164.040,A -90.000,B 90.000,C 0.000} C_DIS
LIN {X 2.703,Y -29.558,Z -163.665,A -90.000,B 90.000,C 0.000} C_DIS
LIN {X 2.535,Y -29.480,Z -163.350,A -90.000,B 90.000,C 0.000} C_DIS
LIN {X 2.356,Y -29.408,Z -163.019,A -90.000,B 90.000,C 0.000} C_DIS
LIN {X 2.261,Y -29.401,Z -162.873,A -90.000,B 90.000,C 0.000} C_DIS
LIN {X 1.852,Y -29.308,Z -162.452,A -90.000,B 90.000,C 0.000} C_DIS
LIN {X 1.852,Y -60.000,Z -162.452,A -90.000,B 90.000,C 0.000} C_DIS
LIN {X -102.050,Y -60.000,Z -243.561,A -90.000,B 90.000,C 0.000} C_DIS
LIN {X -102.050,Y -29.308,Z -243.561,A -90.000,B 90.000,C 0.000} C_DIS
LIN {X -100.659,Y -29.308,Z -242.529,A -90.000,B 90.000,C 0.000} C_DIS
LIN {X -95.849,Y -29.308,Z -239.248,A -90.000,B 90.000,C 0.000} C_DIS
LIN {X -92.915,Y -29.308,Z -237.193,A -90.000,B 90.000,C 0.000} C_DIS
LIN {X -90.063,Y -29.308,Z -235.343,A -90.000,B 90.000,C 0.000} C_DIS
LIN {X -84.434,Y -29.308,Z -231.608,A -90.000,B 90.000,C 0.000} C_DIS
LIN {X -83.569,Y -29.308,Z -231.073,A -90.000,B 90.000,C 0.000} C_DIS
LIN {X -80.135,Y -29.308,Z -228.922,A -90.000,B 90.000,C 0.000} C_DIS
LIN {X -75.991,Y -29.308,Z -226.342,A -90.000,B 90.000,C 0.000} C_DIS
LIN {X -70.108,Y -29.308,Z -222.914,A -90.000,B 90.000,C 0.000} C_DIS
LIN {X -67.329,Y -29.308,Z -221.317,A -90.000,B 90.000,C 0.000} C_DIS
LIN {X -59.222,Y -29.308,Z -216.869,A -90.000,B 90.000,C 0.000} C_DIS
LIN {X -58.840,Y -29.308,Z -216.663,A -90.000,B 90.000,C 0.000} C_DIS
LIN {X -52.926,Y -29.308,Z -213.515,A -90.000,B 90.000,C 0.000} C_DIS
LIN {X -50.896,Y -29.308,Z -212.456,A -90.000,B 90.000,C 0.000} C_DIS
LIN {X -47.193,Y -29.308,Z -210.504,A -90.000,B 90.000,C 0.000} C_DIS
LIN {X -43.851,Y -29.308,Z -208.773,A -90.000,B 90.000,C 0.000} C_DIS
LIN {X -38.065,Y -29.308,Z -205.658,A -90.000,B 90.000,C 0.000} C_DIS
LIN {X -37.545,Y -29.308,Z -205.366,A -90.000,B 90.000,C 0.000} C_DIS
LIN {X -34.672,Y -29.308,Z -203.735,A -90.000,B 90.000,C 0.000} C_DIS
LIN {X -33.528,Y -29.308,Z -203.087,A -90.000,B 90.000,C 0.000} C_DIS
LIN {X -29.580,Y -29.308,Z -200.697,A -90.000,B 90.000,C 0.000} C_DIS
LIN {X -25.997,Y -29.308,Z -198.358,A -90.000,B 90.000,C 0.000} C_DIS
LIN {X -22.969,Y -29.308,Z -196.234,A -90.000,B 90.000,C 0.000} C_DIS
LIN {X -19.780,Y -29.308,Z -193.821,A -90.000,B 90.000,C 0.000} C_DIS
LIN {X -16.589,Y -29.308,Z -191.218,A -90.000,B 90.000,C 0.000} C_DIS
LIN {X -13.561,Y -29.308,Z -188.575,A -90.000,B 90.000,C 0.000} C_DIS
LIN {X -12.176,Y -29.308,Z -187.272,A -90.000,B 90.000,C 0.000} C_DIS
LIN {X -10.317,Y -29.308,Z -185.555,A -90.000,B 90.000,C 0.000} C_DIS
LIN {X -8.519,Y -29.308,Z -183.714,A -90.000,B 90.000,C 0.000} C_DIS
LIN {X -7.045,Y -29.308,Z -182.269,A -90.000,B 90.000,C 0.000} C_DIS
LIN {X -6.501,Y -29.308,Z -181.663,A -90.000,B 90.000,C 0.000} C_DIS
LIN {X -4.186,Y -29.308,Z -179.068,A -90.000,B 90.000,C 0.000} C_DIS
LIN {X -3.472,Y -29.308,Z -178.113,A -90.000,B 90.000,C 0.000} C_DIS
LIN {X -1.865,Y -29.308,Z -176.010,A -90.000,B 90.000,C 0.000} C_DIS
LIN {X -1.690,Y -29.308,Z -175.788,A -90.000,B 90.000,C 0.000} C_DIS
LIN {X -1.632,Y -29.308,Z -175.702,A -90.000,B 90.000,C 0.000} C_DIS
LIN {X -1.325,Y -29.308,Z -175.189,A -90.000,B 90.000,C 0.000} C_DIS
LIN {X -0.089,Y -29.308,Z -173.225,A -90.000,B 90.000,C 0.000} C_DIS
LIN {X 0.298,Y -29.308,Z -172.518,A -90.000,B 90.000,C 0.000} C_DIS
LIN {X 0.550,Y -29.308,Z -171.981,A -90.000,B 90.000,C 0.000} C_DIS
LIN {X 0.884,Y -29.308,Z -171.086,A -90.000,B 90.000,C 0.000} C_DIS
LIN {X 1.747,Y -29.308,Z -168.979,A -90.000,B 90.000,C 0.000} C_DIS
LIN {X 1.754,Y -29.308,Z -168.960,A -90.000,B 90.000,C 0.000} C_DIS
LIN {X 2.054,Y -29.308,Z -167.726,A -90.000,B 90.000,C 0.000} C_DIS
LIN {X 2.385,Y -29.308,Z -165.593,A -90.000,B 90.000,C 0.000} C_DIS
LIN {X 2.291,Y -29.308,Z -164.350,A -90.000,B 90.000,C 0.000} C_DIS
LIN {X 2.242,Y -29.308,Z -163.681,A -90.000,B 90.000,C 0.000} C_DIS
LIN {X 2.163,Y -29.308,Z -163.022,A -90.000,B 90.000,C 0.000} C_DIS
LIN {X 1.765,Y -29.308,Z -162.291,A -90.000,B 90.000,C 0.000} C_DIS
LIN {X 1.143,Y -29.308,Z -161.103,A -90.000,B 90.000,C 0.000} C_DIS
LIN {X 1.004,Y -29.308,Z -160.968,A -90.000,B 90.000,C 0.000} C_DIS
LIN {X 0.095,Y -29.308,Z -160.011,A -90.000,B 90.000,C 0.000} C_DIS
LIN {X -0.163,Y -29.308,Z -159.733,A -90.000,B 90.000,C 0.000} C_DIS
LIN {X -0.360,Y -29.308,Z -159.510,A -90.000,B 90.000,C 0.000} C_DIS
LIN {X -1.822,Y -29.308,Z -158.388,A -90.000,B 90.000,C 0.000} C_DIS
LIN {X -2.239,Y -29.308,Z -158.051,A -90.000,B 90.000,C 0.000} C_DIS
LIN {X -3.624,Y -29.308,Z -157.235,A -90.000,B 90.000,C 0.000} C_DIS
LIN {X -4.589,Y -29.308,Z -156.599,A -90.000,B 90.000,C 0.000} C_DIS
LIN {X -6.558,Y -29.308,Z -155.471,A -90.000,B 90.000,C 0.000} C_DIS
LIN {X -7.083,Y -29.308,Z -155.188,A -90.000,B 90.000,C 0.000} C_DIS
LIN {X -7.746,Y -29.308,Z -154.802,A -90.000,B 90.000,C 0.000} C_DIS
LIN {X -9.613,Y -29.308,Z -153.707,A -90.000,B 90.000,C 0.000} C_DIS
LIN {X -9.711,Y -29.308,Z -153.654,A -90.000,B 90.000,C 0.000} C_DIS
LIN {X -9.949,Y -29.308,Z -153.505,A -90.000,B 90.000,C 0.000} C_DIS
LIN {X -12.007,Y -29.308,Z -152.203,A -90.000,B 90.000,C 0.000} C_DIS
LIN {X -12.443,Y -29.308,Z -151.952,A -90.000,B 90.000,C 0.000} C_DIS
LIN {X -12.845,Y -29.308,Z -151.696,A -90.000,B 90.000,C 0.000} C_DIS
LIN {X -14.301,Y -29.308,Z -150.689,A -90.000,B 90.000,C 0.000} C_DIS
LIN {X -15.780,Y -29.308,Z -149.749,A -90.000,B 90.000,C 0.000} C_DIS
LIN {X -16.172,Y -29.308,Z -149.468,A -90.000,B 90.000,C 0.000} C_DIS
LIN {X -16.662,Y -29.308,Z -149.100,A -90.000,B 90.000,C 0.000} C_DIS
LIN {X -18.399,Y -29.308,Z -147.872,A -90.000,B 90.000,C 0.000} C_DIS
LIN {X -19.357,Y -29.308,Z -147.234,A -90.000,B 90.000,C 0.000} C_DIS
LIN {X -19.837,Y -29.308,Z -146.865,A -90.000,B 90.000,C 0.000} C_DIS
LIN {X -20.632,Y -29.308,Z -146.244,A -90.000,B 90.000,C 0.000} C_DIS
LIN {X -23.002,Y -29.308,Z -144.463,A -90.000,B 90.000,C 0.000} C_DIS
LIN {X -23.257,Y -29.308,Z -144.265,A -90.000,B 90.000,C 0.000} C_DIS
LIN {X -23.386,Y -29.308,Z -144.162,A -90.000,B 90.000,C 0.000} C_DIS
LIN {X -24.407,Y -29.308,Z -143.277,A -90.000,B 90.000,C 0.000} C_DIS
LIN {X -25.887,Y -29.308,Z -142.029,A -90.000,B 90.000,C 0.000} C_DIS
LIN {X -26.771,Y -29.308,Z -141.273,A -90.000,B 90.000,C 0.000} C_DIS
LIN {X -27.123,Y -29.308,Z -140.936,A -90.000,B 90.000,C 0.000} C_DIS
LIN {X -28.241,Y -29.308,Z -139.795,A -90.000,B 90.000,C 0.000} C_DIS
LIN {X -29.251,Y -29.308,Z -138.753,A -90.000,B 90.000,C 0.000} C_DIS
LIN {X -30.308,Y -29.308,Z -137.696,A -90.000,B 90.000,C 0.000} C_DIS
LIN {X -30.623,Y -29.308,Z -137.323,A -90.000,B 90.000,C 0.000} C_DIS
LIN {X -30.739,Y -29.308,Z -137.179,A -90.000,B 90.000,C 0.000} C_DIS
LIN {X -30.985,Y -29.308,Z -136.880,A -90.000,B 90.000,C 0.000} C_DIS
LIN {X -32.999,Y -29.308,Z -134.398,A -90.000,B 90.000,C 0.000} C_DIS
LIN {X -33.264,Y -29.308,Z -134.066,A -90.000,B 90.000,C 0.000} C_DIS
LIN {X -33.542,Y -29.308,Z -133.667,A -90.000,B 90.000,C 0.000} C_DIS
LIN {X -35.008,Y -29.308,Z -131.423,A -90.000,B 90.000,C 0.000} C_DIS
LIN {X -35.793,Y -29.308,Z -130.228,A -90.000,B 90.000,C 0.000} C_DIS
LIN {X -36.028,Y -29.308,Z -129.802,A -90.000,B 90.000,C 0.000} C_DIS
LIN {X -36.754,Y -29.308,Z -128.429,A -90.000,B 90.000,C 0.000} C_DIS
LIN {X -37.821,Y -29.308,Z -126.344,A -90.000,B 90.000,C 0.000} C_DIS
LIN {X -38.023,Y -29.308,Z -125.877,A -90.000,B 90.000,C 0.000} C_DIS
LIN {X -39.000,Y -29.308,Z -123.416,A -90.000,B 90.000,C 0.000} C_DIS
LIN {X -39.428,Y -29.308,Z -122.291,A -90.000,B 90.000,C 0.000} C_DIS
LIN {X -39.583,Y -29.308,Z -121.834,A -90.000,B 90.000,C 0.000} C_DIS
LIN {X -40.313,Y -29.308,Z -119.079,A -90.000,B 90.000,C 0.000} C_DIS
LIN {X -40.501,Y -29.308,Z -118.363,A -90.000,B 90.000,C 0.000} C_DIS
LIN {X -40.581,Y -29.308,Z -118.067,A -90.000,B 90.000,C 0.000} C_DIS
LIN {X -40.778,Y -29.308,Z -117.313,A -90.000,B 90.000,C 0.000} C_DIS
LIN {X -40.872,Y -29.308,Z -116.765,A -90.000,B 90.000,C 0.000} C_DIS
LIN {X -40.919,Y -29.308,Z -116.545,A -90.000,B 90.000,C 0.000} C_DIS
LIN {X -41.283,Y -29.308,Z -114.656,A -90.000,B 90.000,C 0.000} C_DIS
LIN {X -41.349,Y -29.308,Z -114.333,A -90.000,B 90.000,C 0.000} C_DIS
LIN {X -41.570,Y -29.308,Z -113.433,A -90.000,B 90.000,C 0.000} C_DIS
LIN {X -41.728,Y -29.308,Z -112.873,A -90.000,B 90.000,C 0.000} C_DIS
LIN {X -41.934,Y -29.308,Z -112.280,A -90.000,B 90.000,C 0.000} C_DIS
LIN {X -42.261,Y -29.308,Z -111.491,A -90.000,B 90.000,C 0.000} C_DIS
LIN {X -42.489,Y -29.308,Z -111.024,A -90.000,B 90.000,C 0.000} C_DIS
LIN {X -43.178,Y -29.308,Z -109.808,A -90.000,B 90.000,C 0.000} C_DIS
LIN {X -43.317,Y -29.308,Z -109.588,A -90.000,B 90.000,C 0.000} C_DIS
LIN {X -44.605,Y -29.308,Z -107.753,A -90.000,B 90.000,C 0.000} C_DIS
LIN {X -44.951,Y -29.308,Z -107.304,A -90.000,B 90.000,C 0.000} C_DIS
LIN {X -46.157,Y -29.308,Z -105.659,A -90.000,B 90.000,C 0.000} C_DIS
LIN {X -46.573,Y -29.308,Z -105.148,A -90.000,B 90.000,C 0.000} C_DIS
LIN {X -47.770,Y -29.308,Z -103.591,A -90.000,B 90.000,C 0.000} C_DIS
LIN {X -48.810,Y -29.308,Z -102.339,A -90.000,B 90.000,C 0.000} C_DIS
LIN {X -49.040,Y -29.308,Z -102.039,A -90.000,B 90.000,C 0.000} C_DIS
LIN {X -49.241,Y -29.308,Z -101.793,A -90.000,B 90.000,C 0.000} C_DIS
LIN {X -51.149,Y -29.308,Z -99.417,A -90.000,B 90.000,C 0.000} C_DIS
LIN {X -52.682,Y -29.308,Z -97.266,A -90.000,B 90.000,C 0.000} C_DIS
LIN {X -53.359,Y -29.308,Z -96.353,A -90.000,B 90.000,C 0.000} C_DIS
LIN {X -54.196,Y -29.308,Z -95.147,A -90.000,B 90.000,C 0.000} C_DIS
LIN {X -55.538,Y -29.308,Z -93.285,A -90.000,B 90.000,C 0.000} C_DIS
LIN {X -55.693,Y -29.308,Z -93.062,A -90.000,B 90.000,C 0.000} C_DIS
LIN {X -56.045,Y -29.308,Z -92.576,A -90.000,B 90.000,C 0.000} C_DIS
LIN {X -57.446,Y -29.308,Z -90.556,A -90.000,B 90.000,C 0.000} C_DIS
LIN {X -57.624,Y -29.308,Z -90.278,A -90.000,B 90.000,C 0.000} C_DIS
LIN {X -58.614,Y -29.308,Z -88.789,A -90.000,B 90.000,C 0.000} C_DIS
LIN {X -59.481,Y -29.308,Z -87.470,A -90.000,B 90.000,C 0.000} C_DIS
LIN {X -60.164,Y -29.308,Z -86.512,A -90.000,B 90.000,C 0.000} C_DIS
LIN {X -61.210,Y -29.308,Z -85.139,A -90.000,B 90.000,C 0.000} C_DIS
LIN {X -61.992,Y -29.308,Z -84.183,A -90.000,B 90.000,C 0.000} C_DIS
LIN {X -62.830,Y -29.308,Z -83.065,A -90.000,B 90.000,C 0.000} C_DIS
LIN {X -63.070,Y -29.308,Z -82.755,A -90.000,B 90.000,C 0.000} C_DIS
LIN {X -63.276,Y -29.308,Z -82.471,A -90.000,B 90.000,C 0.000} C_DIS
LIN {X -63.911,Y -29.308,Z -81.582,A -90.000,B 90.000,C 0.000} C_DIS
LIN {X -64.489,Y -29.308,Z -80.863,A -90.000,B 90.000,C 0.000} C_DIS
LIN {X -64.824,Y -29.308,Z -80.406,A -90.000,B 90.000,C 0.000} C_DIS
LIN {X -65.513,Y -29.308,Z -79.574,A -90.000,B 90.000,C 0.000} C_DIS
LIN {X -66.220,Y -29.308,Z -78.603,A -90.000,B 90.000,C 0.000} C_DIS
LIN {X -67.877,Y -29.308,Z -76.169,A -90.000,B 90.000,C 0.000} C_DIS
LIN {X -68.903,Y -29.308,Z -74.564,A -90.000,B 90.000,C 0.000} C_DIS
LIN {X -69.308,Y -29.308,Z -73.952,A -90.000,B 90.000,C 0.000} C_DIS
LIN {X -69.820,Y -29.308,Z -73.273,A -90.000,B 90.000,C 0.000} C_DIS
LIN {X -70.184,Y -29.308,Z -72.827,A -90.000,B 90.000,C 0.000} C_DIS
LIN {X -70.760,Y -29.308,Z -72.102,A -90.000,B 90.000,C 0.000} C_DIS
LIN {X -72.178,Y -29.308,Z -70.694,A -90.000,B 90.000,C 0.000} C_DIS
LIN {X -72.224,Y -29.308,Z -70.649,A -90.000,B 90.000,C 0.000} C_DIS
LIN {X -72.642,Y -29.308,Z -70.285,A -90.000,B 90.000,C 0.000} C_DIS
LIN {X -73.359,Y -29.308,Z -69.762,A -90.000,B 90.000,C 0.000} C_DIS
LIN {X -73.386,Y -29.308,Z -69.741,A -90.000,B 90.000,C 0.000} C_DIS
LIN {X -73.983,Y -29.308,Z -69.351,A -90.000,B 90.000,C 0.000} C_DIS
LIN {X -74.194,Y -29.308,Z -69.227,A -90.000,B 90.000,C 0.000} C_DIS
LIN {X -74.496,Y -29.308,Z -69.103,A -90.000,B 90.000,C 0.000} C_DIS
LIN {X -74.639,Y -29.308,Z -69.049,A -90.000,B 90.000,C 0.000} C_DIS
LIN {X -74.842,Y -29.308,Z -69.031,A -90.000,B 90.000,C 0.000} C_DIS
LIN {X -75.073,Y -29.308,Z -69.069,A -90.000,B 90.000,C 0.000} C_DIS
LIN {X -75.243,Y -29.308,Z -69.093,A -90.000,B 90.000,C 0.000} C_DIS
LIN {X -75.577,Y -29.308,Z -69.204,A -90.000,B 90.000,C 0.000} C_DIS
LIN {X -75.633,Y -29.308,Z -69.220,A -90.000,B 90.000,C 0.000} C_DIS
LIN {X -75.813,Y -29.308,Z -69.297,A -90.000,B 90.000,C 0.000} C_DIS
LIN {X -76.073,Y -29.308,Z -69.398,A -90.000,B 90.000,C 0.000} C_DIS
LIN {X -76.595,Y -29.308,Z -69.566,A -90.000,B 90.000,C 0.000} C_DIS
LIN {X -76.818,Y -29.308,Z -69.621,A -90.000,B 90.000,C 0.000} C_DIS
LIN {X -77.130,Y -29.308,Z -69.689,A -90.000,B 90.000,C 0.000} C_DIS
LIN {X -77.390,Y -29.308,Z -69.734,A -90.000,B 90.000,C 0.000} C_DIS
LIN {X -77.637,Y -29.308,Z -69.769,A -90.000,B 90.000,C 0.000} C_DIS
LIN {X -77.967,Y -29.308,Z -69.787,A -90.000,B 90.000,C 0.000} C_DIS
LIN {X -78.431,Y -29.308,Z -69.777,A -90.000,B 90.000,C 0.000} C_DIS
LIN {X -78.778,Y -29.308,Z -69.745,A -90.000,B 90.000,C 0.000} C_DIS
LIN {X -79.117,Y -29.308,Z -69.664,A -90.000,B 90.000,C 0.000} C_DIS
LIN {X -79.541,Y -29.308,Z -69.536,A -90.000,B 90.000,C 0.000} C_DIS
LIN {X -79.868,Y -29.308,Z -69.408,A -90.000,B 90.000,C 0.000} C_DIS
LIN {X -80.173,Y -29.308,Z -69.234,A -90.000,B 90.000,C 0.000} C_DIS
LIN {X -80.550,Y -29.308,Z -68.954,A -90.000,B 90.000,C 0.000} C_DIS
LIN {X -80.828,Y -29.308,Z -68.739,A -90.000,B 90.000,C 0.000} C_DIS
LIN {X -80.865,Y -29.308,Z -68.705,A -90.000,B 90.000,C 0.000} C_DIS
LIN {X -81.112,Y -29.308,Z -68.450,A -90.000,B 90.000,C 0.000} C_DIS
LIN {X -81.204,Y -29.308,Z -68.343,A -90.000,B 90.000,C 0.000} C_DIS
LIN {X -81.417,Y -29.308,Z -68.047,A -90.000,B 90.000,C 0.000} C_DIS
LIN {X -81.727,Y -29.308,Z -67.575,A -90.000,B 90.000,C 0.000} C_DIS
LIN {X -81.896,Y -29.308,Z -67.254,A -90.000,B 90.000,C 0.000} C_DIS
LIN {X -81.988,Y -29.308,Z -67.066,A -90.000,B 90.000,C 0.000} C_DIS
LIN {X -82.185,Y -29.308,Z -66.525,A -90.000,B 90.000,C 0.000} C_DIS
LIN {X -82.221,Y -29.308,Z -66.413,A -90.000,B 90.000,C 0.000} C_DIS
LIN {X -82.302,Y -29.308,Z -66.145,A -90.000,B 90.000,C 0.000} C_DIS
LIN {X -82.411,Y -29.308,Z -65.838,A -90.000,B 90.000,C 0.000} C_DIS
LIN {X -82.467,Y -29.308,Z -65.687,A -90.000,B 90.000,C 0.000} C_DIS
LIN {X -82.502,Y -29.308,Z -65.567,A -90.000,B 90.000,C 0.000} C_DIS
LIN {X -82.553,Y -29.308,Z -65.421,A -90.000,B 90.000,C 0.000} C_DIS
LIN {X -82.588,Y -29.308,Z -65.339,A -90.000,B 90.000,C 0.000} C_DIS
LIN {X -82.726,Y -29.308,Z -65.030,A -90.000,B 90.000,C 0.000} C_DIS
LIN {X -82.936,Y -29.308,Z -64.520,A -90.000,B 90.000,C 0.000} C_DIS
LIN {X -83.027,Y -29.308,Z -64.293,A -90.000,B 90.000,C 0.000} C_DIS
LIN {X -83.195,Y -29.308,Z -63.767,A -90.000,B 90.000,C 0.000} C_DIS
LIN {X -83.237,Y -29.308,Z -63.614,A -90.000,B 90.000,C 0.000} C_DIS
LIN {X -83.287,Y -29.308,Z -63.390,A -90.000,B 90.000,C 0.000} C_DIS
LIN {X -83.364,Y -29.308,Z -62.978,A -90.000,B 90.000,C 0.000} C_DIS
LIN {X -83.389,Y -29.308,Z -62.793,A -90.000,B 90.000,C 0.000} C_DIS
LIN {X -83.454,Y -29.308,Z -62.265,A -90.000,B 90.000,C 0.000} C_DIS
LIN {X -83.484,Y -29.308,Z -62.052,A -90.000,B 90.000,C 0.000} C_DIS
LIN {X -83.536,Y -29.308,Z -61.778,A -90.000,B 90.000,C 0.000} C_DIS
LIN {X -83.567,Y -29.308,Z -61.489,A -90.000,B 90.000,C 0.000} C_DIS
LIN {X -83.619,Y -29.308,Z -61.201,A -90.000,B 90.000,C 0.000} C_DIS
LIN {X -83.798,Y -29.308,Z -60.652,A -90.000,B 90.000,C 0.000} C_DIS
LIN {X -83.805,Y -29.308,Z -60.627,A -90.000,B 90.000,C 0.000} C_DIS
LIN {X -84.046,Y -29.308,Z -60.123,A -90.000,B 90.000,C 0.000} C_DIS
LIN {X -84.182,Y -29.308,Z -59.795,A -90.000,B 90.000,C 0.000} C_DIS
LIN {X -84.358,Y -29.308,Z -59.481,A -90.000,B 90.000,C 0.000} C_DIS
LIN {X -84.837,Y -29.308,Z -58.578,A -90.000,B 90.000,C 0.000} C_DIS
LIN {X -85.210,Y -29.308,Z -57.933,A -90.000,B 90.000,C 0.000} C_DIS
LIN {X -85.343,Y -29.308,Z -57.685,A -90.000,B 90.000,C 0.000} C_DIS
LIN {X -85.738,Y -29.308,Z -56.884,A -90.000,B 90.000,C 0.000} C_DIS
LIN {X -86.011,Y -29.308,Z -56.262,A -90.000,B 90.000,C 0.000} C_DIS
LIN {X -86.022,Y -29.308,Z -56.237,A -90.000,B 90.000,C 0.000} C_DIS
LIN {X -86.100,Y -29.308,Z -56.014,A -90.000,B 90.000,C 0.000} C_DIS
LIN {X -86.102,Y -29.308,Z -56.000,A -90.000,B 90.000,C 0.000} C_DIS
LIN {X -86.253,Y -29.308,Z -55.463,A -90.000,B 90.000,C 0.000} C_DIS
LIN {X -86.283,Y -29.308,Z -55.227,A -90.000,B 90.000,C 0.000} C_DIS
LIN {X -86.283,Y -29.308,Z -55.107,A -90.000,B 90.000,C 0.000} C_DIS
LIN {X -86.321,Y -29.308,Z -54.753,A -90.000,B 90.000,C 0.000} C_DIS
LIN {X -86.298,Y -29.308,Z -54.344,A -90.000,B 90.000,C 0.000} C_DIS
LIN {X -86.269,Y -29.308,Z -54.104,A -90.000,B 90.000,C 0.000} C_DIS
LIN {X -86.230,Y -29.308,Z -53.929,A -90.000,B 90.000,C 0.000} C_DIS
LIN {X -86.168,Y -29.308,Z -53.790,A -90.000,B 90.000,C 0.000} C_DIS
LIN {X -86.082,Y -29.308,Z -53.633,A -90.000,B 90.000,C 0.000} C_DIS
LIN {X -85.957,Y -29.308,Z -53.505,A -90.000,B 90.000,C 0.000} C_DIS
LIN {X -85.550,Y -29.308,Z -53.277,A -90.000,B 90.000,C 0.000} C_DIS
LIN {X -85.368,Y -29.308,Z -53.180,A -90.000,B 90.000,C 0.000} C_DIS
LIN {X -85.152,Y -29.308,Z -53.081,A -90.000,B 90.000,C 0.000} C_DIS
LIN {X -85.138,Y -29.308,Z -53.076,A -90.000,B 90.000,C 0.000} C_DIS
LIN {X -84.907,Y -29.308,Z -53.024,A -90.000,B 90.000,C 0.000} C_DIS
LIN {X -84.627,Y -29.308,Z -53.021,A -90.000,B 90.000,C 0.000} C_DIS
LIN {X -84.602,Y -29.308,Z -53.023,A -90.000,B 90.000,C 0.000} C_DIS
LIN {X -83.793,Y -29.308,Z -53.148,A -90.000,B 90.000,C 0.000} C_DIS
LIN {X -83.520,Y -29.308,Z -53.216,A -90.000,B 90.000,C 0.000} C_DIS
LIN {X -82.901,Y -29.308,Z -53.385,A -90.000,B 90.000,C 0.000} C_DIS
LIN {X -82.607,Y -29.308,Z -53.469,A -90.000,B 90.000,C 0.000} C_DIS
LIN {X -82.260,Y -29.308,Z -53.575,A -90.000,B 90.000,C 0.000} C_DIS
LIN {X -82.167,Y -29.308,Z -53.614,A -90.000,B 90.000,C 0.000} C_DIS
LIN {X -81.991,Y -29.308,Z -53.693,A -90.000,B 90.000,C 0.000} C_DIS
LIN {X -81.010,Y -29.308,Z -54.146,A -90.000,B 90.000,C 0.000} C_DIS
LIN {X -80.181,Y -29.308,Z -54.602,A -90.000,B 90.000,C 0.000} C_DIS
LIN {X -80.023,Y -29.308,Z -54.700,A -90.000,B 90.000,C 0.000} C_DIS
LIN {X -78.692,Y -29.308,Z -55.627,A -90.000,B 90.000,C 0.000} C_DIS
LIN {X -78.411,Y -29.308,Z -55.839,A -90.000,B 90.000,C 0.000} C_DIS
LIN {X -78.296,Y -29.308,Z -55.936,A -90.000,B 90.000,C 0.000} C_DIS
LIN {X -77.163,Y -29.308,Z -56.798,A -90.000,B 90.000,C 0.000} C_DIS
LIN {X -76.756,Y -29.308,Z -57.139,A -90.000,B 90.000,C 0.000} C_DIS
LIN {X -76.357,Y -29.308,Z -57.383,A -90.000,B 90.000,C 0.000} C_DIS
LIN {X -76.173,Y -29.308,Z -57.509,A -90.000,B 90.000,C 0.000} C_DIS
LIN {X -75.781,Y -29.308,Z -57.673,A -90.000,B 90.000,C 0.000} C_DIS
LIN {X -75.668,Y -29.308,Z -57.728,A -90.000,B 90.000,C 0.000} C_DIS
LIN {X -75.074,Y -29.308,Z -57.884,A -90.000,B 90.000,C 0.000} C_DIS
LIN {X -74.895,Y -29.308,Z -57.941,A -90.000,B 90.000,C 0.000} C_DIS
LIN {X -74.819,Y -29.308,Z -57.950,A -90.000,B 90.000,C 0.000} C_DIS
LIN {X -73.695,Y -29.308,Z -58.054,A -90.000,B 90.000,C 0.000} C_DIS
LIN {X -73.250,Y -29.308,Z -58.051,A -90.000,B 90.000,C 0.000} C_DIS
LIN {X -72.096,Y -29.308,Z -57.889,A -90.000,B 90.000,C 0.000} C_DIS
LIN {X -71.132,Y -29.308,Z -57.766,A -90.000,B 90.000,C 0.000} C_DIS
LIN {X -70.465,Y -29.308,Z -57.615,A -90.000,B 90.000,C 0.000} C_DIS
LIN {X -69.608,Y -29.308,Z -57.448,A -90.000,B 90.000,C 0.000} C_DIS
LIN {X -68.653,Y -29.308,Z -57.215,A -90.000,B 90.000,C 0.000} C_DIS
LIN {X -67.391,Y -29.308,Z -56.810,A -90.000,B 90.000,C 0.000} C_DIS
LIN {X -67.137,Y -29.308,Z -56.710,A -90.000,B 90.000,C 0.000} C_DIS
LIN {X -66.052,Y -29.308,Z -56.358,A -90.000,B 90.000,C 0.000} C_DIS
LIN {X -65.482,Y -29.308,Z -56.132,A -90.000,B 90.000,C 0.000} C_DIS
LIN {X -64.851,Y -29.308,Z -55.889,A -90.000,B 90.000,C 0.000} C_DIS
LIN {X -63.760,Y -29.308,Z -55.413,A -90.000,B 90.000,C 0.000} C_DIS
LIN {X -62.088,Y -29.308,Z -54.821,A -90.000,B 90.000,C 0.000} C_DIS
LIN {X -60.476,Y -29.308,Z -54.401,A -90.000,B 90.000,C 0.000} C_DIS
LIN {X -60.277,Y -29.308,Z -54.357,A -90.000,B 90.000,C 0.000} C_DIS
LIN {X -59.975,Y -29.308,Z -54.309,A -90.000,B 90.000,C 0.000} C_DIS
LIN {X -58.448,Y -29.308,Z -54.158,A -90.000,B 90.000,C 0.000} C_DIS
LIN {X -57.234,Y -29.308,Z -54.106,A -90.000,B 90.000,C 0.000} C_DIS
LIN {X -55.540,Y -29.308,Z -54.135,A -90.000,B 90.000,C 0.000} C_DIS
LIN {X -54.330,Y -29.308,Z -54.194,A -90.000,B 90.000,C 0.000} C_DIS
LIN {X -53.511,Y -29.308,Z -54.246,A -90.000,B 90.000,C 0.000} C_DIS
LIN {X -53.193,Y -29.308,Z -54.273,A -90.000,B 90.000,C 0.000} C_DIS
LIN {X -51.223,Y -29.308,Z -54.509,A -90.000,B 90.000,C 0.000} C_DIS
LIN {X -50.881,Y -29.308,Z -54.553,A -90.000,B 90.000,C 0.000} C_DIS
LIN {X -48.137,Y -29.308,Z -54.941,A -90.000,B 90.000,C 0.000} C_DIS
LIN {X -46.120,Y -29.308,Z -55.320,A -90.000,B 90.000,C 0.000} C_DIS
LIN {X -43.370,Y -29.308,Z -55.918,A -90.000,B 90.000,C 0.000} C_DIS
LIN {X -41.703,Y -29.308,Z -56.310,A -90.000,B 90.000,C 0.000} C_DIS
LIN {X -38.030,Y -29.308,Z -57.209,A -90.000,B 90.000,C 0.000} C_DIS
LIN {X -36.355,Y -29.308,Z -57.615,A -90.000,B 90.000,C 0.000} C_DIS
LIN {X -35.314,Y -29.308,Z -57.840,A -90.000,B 90.000,C 0.000} C_DIS
LIN {X -34.576,Y -29.308,Z -57.955,A -90.000,B 90.000,C 0.000} C_DIS
LIN {X -32.395,Y -29.308,Z -58.194,A -90.000,B 90.000,C 0.000} C_DIS
LIN {X -29.664,Y -29.308,Z -58.541,A -90.000,B 90.000,C 0.000} C_DIS
LIN {X -28.228,Y -29.308,Z -58.715,A -90.000,B 90.000,C 0.000} C_DIS
LIN {X -27.180,Y -29.308,Z -58.860,A -90.000,B 90.000,C 0.000} C_DIS
LIN {X -25.794,Y -29.308,Z -58.982,A -90.000,B 90.000,C 0.000} C_DIS
LIN {X -25.319,Y -29.308,Z -59.031,A -90.000,B 90.000,C 0.000} C_DIS
LIN {X -24.289,Y -29.308,Z -59.027,A -90.000,B 90.000,C 0.000} C_DIS
LIN {X -23.894,Y -29.308,Z -59.045,A -90.000,B 90.000,C 0.000} C_DIS
LIN {X -23.530,Y -29.308,Z -58.984,A -90.000,B 90.000,C 0.000} C_DIS
LIN {X -22.931,Y -29.308,Z -58.928,A -90.000,B 90.000,C 0.000} C_DIS
LIN {X -22.654,Y -29.308,Z -58.830,A -90.000,B 90.000,C 0.000} C_DIS
LIN {X -22.187,Y -29.308,Z -58.705,A -90.000,B 90.000,C 0.000} C_DIS
LIN {X -22.053,Y -29.308,Z -58.636,A -90.000,B 90.000,C 0.000} C_DIS
LIN {X -21.305,Y -29.308,Z -58.317,A -90.000,B 90.000,C 0.000} C_DIS
LIN {X -21.163,Y -29.308,Z -58.232,A -90.000,B 90.000,C 0.000} C_DIS
LIN {X -19.091,Y -29.308,Z -57.103,A -90.000,B 90.000,C 0.000} C_DIS
LIN {X -18.992,Y -29.308,Z -57.050,A -90.000,B 90.000,C 0.000} C_DIS
LIN {X -17.751,Y -29.308,Z -56.481,A -90.000,B 90.000,C 0.000} C_DIS
LIN {X -16.945,Y -29.308,Z -56.142,A -90.000,B 90.000,C 0.000} C_DIS
LIN {X -16.552,Y -29.308,Z -55.986,A -90.000,B 90.000,C 0.000} C_DIS
LIN {X -14.526,Y -29.308,Z -55.387,A -90.000,B 90.000,C 0.000} C_DIS
LIN {X -14.117,Y -29.308,Z -55.278,A -90.000,B 90.000,C 0.000} C_DIS
LIN {X -13.753,Y -29.308,Z -55.189,A -90.000,B 90.000,C 0.000} C_DIS
LIN {X -13.576,Y -29.308,Z -55.148,A -90.000,B 90.000,C 0.000} C_DIS
LIN {X -13.345,Y -29.308,Z -55.115,A -90.000,B 90.000,C 0.000} C_DIS
LIN {X -12.545,Y -29.308,Z -55.032,A -90.000,B 90.000,C 0.000} C_DIS
LIN {X -11.451,Y -29.308,Z -54.978,A -90.000,B 90.000,C 0.000} C_DIS
LIN {X -10.294,Y -29.308,Z -54.903,A -90.000,B 90.000,C 0.000} C_DIS
LIN {X -9.729,Y -29.308,Z -54.905,A -90.000,B 90.000,C 0.000} C_DIS
LIN {X -9.578,Y -29.308,Z -54.908,A -90.000,B 90.000,C 0.000} C_DIS
LIN {X -9.342,Y -29.308,Z -54.921,A -90.000,B 90.000,C 0.000} C_DIS
LIN {X -8.355,Y -29.308,Z -55.042,A -90.000,B 90.000,C 0.000} C_DIS
LIN {X -7.679,Y -29.308,Z -55.133,A -90.000,B 90.000,C 0.000} C_DIS
LIN {X -7.280,Y -29.308,Z -55.191,A -90.000,B 90.000,C 0.000} C_DIS
LIN {X -6.863,Y -29.308,Z -55.260,A -90.000,B 90.000,C 0.000} C_DIS
LIN {X -6.490,Y -29.308,Z -55.330,A -90.000,B 90.000,C 0.000} C_DIS
LIN {X -4.215,Y -29.308,Z -55.882,A -90.000,B 90.000,C 0.000} C_DIS
LIN {X -1.838,Y -29.308,Z -56.578,A -90.000,B 90.000,C 0.000} C_DIS
LIN {X -0.973,Y -29.308,Z -56.836,A -90.000,B 90.000,C 0.000} C_DIS
LIN {X 0.608,Y -29.308,Z -57.303,A -90.000,B 90.000,C 0.000} C_DIS
LIN {X 1.264,Y -29.308,Z -57.478,A -90.000,B 90.000,C 0.000} C_DIS
LIN {X 3.041,Y -29.308,Z -57.932,A -90.000,B 90.000,C 0.000} C_DIS
LIN {X 4.643,Y -29.308,Z -58.201,A -90.000,B 90.000,C 0.000} C_DIS
LIN {X 4.898,Y -29.308,Z -58.243,A -90.000,B 90.000,C 0.000} C_DIS
LIN {X 4.968,Y -29.308,Z -58.250,A -90.000,B 90.000,C 0.000} C_DIS
LIN {X 6.293,Y -29.308,Z -58.352,A -90.000,B 90.000,C 0.000} C_DIS
LIN {X 6.943,Y -29.308,Z -58.362,A -90.000,B 90.000,C 0.000} C_DIS
LIN {X 7.658,Y -29.308,Z -58.360,A -90.000,B 90.000,C 0.000} C_DIS
LIN {X 8.615,Y -29.308,Z -58.308,A -90.000,B 90.000,C 0.000} C_DIS
LIN {X 8.888,Y -29.308,Z -58.287,A -90.000,B 90.000,C 0.000} C_DIS
LIN {X 9.972,Y -29.308,Z -58.200,A -90.000,B 90.000,C 0.000} C_DIS
LIN {X 10.948,Y -29.308,Z -58.139,A -90.000,B 90.000,C 0.000} C_DIS
LIN {X 11.107,Y -29.308,Z -58.124,A -90.000,B 90.000,C 0.000} C_DIS
LIN {X 11.426,Y -29.308,Z -58.099,A -90.000,B 90.000,C 0.000} C_DIS
LIN {X 12.056,Y -29.308,Z -58.061,A -90.000,B 90.000,C 0.000} C_DIS
LIN {X 12.258,Y -29.308,Z -58.030,A -90.000,B 90.000,C 0.000} C_DIS
LIN {X 12.960,Y -29.308,Z -57.969,A -90.000,B 90.000,C 0.000} C_DIS
LIN {X 13.028,Y -29.308,Z -57.954,A -90.000,B 90.000,C 0.000} C_DIS
LIN {X 13.316,Y -29.308,Z -57.915,A -90.000,B 90.000,C 0.000} C_DIS
LIN {X 13.534,Y -29.308,Z -57.887,A -90.000,B 90.000,C 0.000} C_DIS
LIN {X 13.953,Y -29.308,Z -57.789,A -90.000,B 90.000,C 0.000} C_DIS
LIN {X 14.128,Y -29.308,Z -57.761,A -90.000,B 90.000,C 0.000} C_DIS
LIN {X 14.407,Y -29.308,Z -57.687,A -90.000,B 90.000,C 0.000} C_DIS
LIN {X 14.771,Y -29.308,Z -57.629,A -90.000,B 90.000,C 0.000} C_DIS
LIN {X 14.874,Y -29.308,Z -57.614,A -90.000,B 90.000,C 0.000} C_DIS
LIN {X 15.147,Y -29.308,Z -57.544,A -90.000,B 90.000,C 0.000} C_DIS
LIN {X 15.558,Y -29.308,Z -57.486,A -90.000,B 90.000,C 0.000} C_DIS
LIN {X 15.990,Y -29.308,Z -57.460,A -90.000,B 90.000,C 0.000} C_DIS
LIN {X 16.224,Y -29.308,Z -57.427,A -90.000,B 90.000,C 0.000} C_DIS
LIN {X 16.647,Y -29.308,Z -57.417,A -90.000,B 90.000,C 0.000} C_DIS
LIN {X 17.186,Y -29.308,Z -57.462,A -90.000,B 90.000,C 0.000} C_DIS
LIN {X 17.264,Y -29.308,Z -57.461,A -90.000,B 90.000,C 0.000} C_DIS
LIN {X 17.686,Y -29.308,Z -57.502,A -90.000,B 90.000,C 0.000} C_DIS
LIN {X 18.100,Y -29.308,Z -57.591,A -90.000,B 90.000,C 0.000} C_DIS
LIN {X 18.644,Y -29.308,Z -57.741,A -90.000,B 90.000,C 0.000} C_DIS
LIN {X 18.688,Y -29.308,Z -57.751,A -90.000,B 90.000,C 0.000} C_DIS
LIN {X 19.056,Y -29.308,Z -57.877,A -90.000,B 90.000,C 0.000} C_DIS
LIN {X 19.151,Y -29.308,Z -57.851,A -90.000,B 90.000,C 0.000} C_DIS
LIN {X 19.383,Y -29.308,Z -57.790,A -90.000,B 90.000,C 0.000} C_DIS
LIN {X 19.459,Y -29.308,Z -57.756,A -90.000,B 90.000,C 0.000} C_DIS
LIN {X 19.594,Y -29.308,Z -57.705,A -90.000,B 90.000,C 0.000} C_DIS
LIN {X 20.022,Y -29.308,Z -57.549,A -90.000,B 90.000,C 0.000} C_DIS
LIN {X 20.464,Y -29.308,Z -57.441,A -90.000,B 90.000,C 0.000} C_DIS
LIN {X 20.816,Y -29.308,Z -57.391,A -90.000,B 90.000,C 0.000} C_DIS
LIN {X 20.940,Y -29.308,Z -57.375,A -90.000,B 90.000,C 0.000} C_DIS
LIN {X 21.379,Y -29.308,Z -57.343,A -90.000,B 90.000,C 0.000} C_DIS
LIN {X 21.448,Y -29.308,Z -57.345,A -90.000,B 90.000,C 0.000} C_DIS
LIN {X 21.649,Y -29.308,Z -57.212,A -90.000,B 90.000,C 0.000} C_DIS
LIN {X 22.422,Y -29.308,Z -56.755,A -90.000,B 90.000,C 0.000} C_DIS
LIN {X 22.658,Y -29.308,Z -56.617,A -90.000,B 90.000,C 0.000} C_DIS
LIN {X 22.710,Y -29.308,Z -56.325,A -90.000,B 90.000,C 0.000} C_DIS
LIN {X 22.737,Y -29.308,Z -56.192,A -90.000,B 90.000,C 0.000} C_DIS
LIN {X 22.772,Y -29.308,Z -56.078,A -90.000,B 90.000,C 0.000} C_DIS
LIN {X 22.861,Y -29.308,Z -55.799,A -90.000,B 90.000,C 0.000} C_DIS
LIN {X 23.006,Y -29.308,Z -55.434,A -90.000,B 90.000,C 0.000} C_DIS
LIN {X 23.185,Y -29.308,Z -55.085,A -90.000,B 90.000,C 0.000} C_DIS
LIN {X 23.229,Y -29.308,Z -55.021,A -90.000,B 90.000,C 0.000} C_DIS
LIN {X 23.354,Y -29.308,Z -54.805,A -90.000,B 90.000,C 0.000} C_DIS
LIN {X 23.594,Y -29.308,Z -54.457,A -90.000,B 90.000,C 0.000} C_DIS
LIN {X 24.081,Y -29.308,Z -53.902,A -90.000,B 90.000,C 0.000} C_DIS
LIN {X 24.401,Y -29.308,Z -53.601,A -90.000,B 90.000,C 0.000} C_DIS
LIN {X 24.554,Y -29.308,Z -53.465,A -90.000,B 90.000,C 0.000} C_DIS
LIN {X 24.908,Y -29.308,Z -53.178,A -90.000,B 90.000,C 0.000} C_DIS
LIN {X 24.955,Y -29.308,Z -53.143,A -90.000,B 90.000,C 0.000} C_DIS
LIN {X 25.043,Y -29.308,Z -53.073,A -90.000,B 90.000,C 0.000} C_DIS
LIN {X 25.440,Y -29.308,Z -52.815,A -90.000,B 90.000,C 0.000} C_DIS
LIN {X 25.450,Y -29.308,Z -52.593,A -90.000,B 90.000,C 0.000} C_DIS
LIN {X 25.526,Y -29.308,Z -52.166,A -90.000,B 90.000,C 0.000} C_DIS
LIN {X 25.622,Y -29.308,Z -51.762,A -90.000,B 90.000,C 0.000} C_DIS
LIN {X 25.655,Y -29.308,Z -51.657,A -90.000,B 90.000,C 0.000} C_DIS
LIN {X 25.714,Y -29.308,Z -51.434,A -90.000,B 90.000,C 0.000} C_DIS
LIN {X 25.753,Y -29.308,Z -51.317,A -90.000,B 90.000,C 0.000} C_DIS
LIN {X 25.880,Y -29.308,Z -50.967,A -90.000,B 90.000,C 0.000} C_DIS
LIN {X 26.066,Y -29.308,Z -50.525,A -90.000,B 90.000,C 0.000} C_DIS
LIN {X 26.196,Y -29.308,Z -50.246,A -90.000,B 90.000,C 0.000} C_DIS
LIN {X 26.291,Y -29.308,Z -50.048,A -90.000,B 90.000,C 0.000} C_DIS
LIN {X 26.629,Y -29.308,Z -49.412,A -90.000,B 90.000,C 0.000} C_DIS
LIN {X 26.899,Y -29.308,Z -48.976,A -90.000,B 90.000,C 0.000} C_DIS
LIN {X 26.977,Y -29.308,Z -48.851,A -90.000,B 90.000,C 0.000} C_DIS
LIN {X 27.214,Y -29.308,Z -48.508,A -90.000,B 90.000,C 0.000} C_DIS
LIN {X 27.357,Y -29.308,Z -48.334,A -90.000,B 90.000,C 0.000} C_DIS
LIN {X 27.637,Y -29.308,Z -48.005,A -90.000,B 90.000,C 0.000} C_DIS
LIN {X 28.103,Y -29.308,Z -47.476,A -90.000,B 90.000,C 0.000} C_DIS
LIN {X 28.429,Y -29.308,Z -47.171,A -90.000,B 90.000,C 0.000} C_DIS
LIN {X 28.887,Y -29.308,Z -46.802,A -90.000,B 90.000,C 0.000} C_DIS
LIN {X 29.157,Y -29.308,Z -46.626,A -90.000,B 90.000,C 0.000} C_DIS
LIN {X 29.540,Y -29.308,Z -46.348,A -90.000,B 90.000,C 0.000} C_DIS
LIN {X 29.923,Y -29.308,Z -46.103,A -90.000,B 90.000,C 0.000} C_DIS
LIN {X 30.457,Y -29.308,Z -45.825,A -90.000,B 90.000,C 0.000} C_DIS
LIN {X 30.886,Y -29.308,Z -45.639,A -90.000,B 90.000,C 0.000} C_DIS
LIN {X 31.387,Y -29.308,Z -45.461,A -90.000,B 90.000,C 0.000} C_DIS
LIN {X 31.833,Y -29.308,Z -45.322,A -90.000,B 90.000,C 0.000} C_DIS
LIN {X 32.264,Y -29.308,Z -45.192,A -90.000,B 90.000,C 0.000} C_DIS
LIN {X 32.822,Y -29.308,Z -45.074,A -90.000,B 90.000,C 0.000} C_DIS
LIN {X 33.293,Y -29.308,Z -44.997,A -90.000,B 90.000,C 0.000} C_DIS
LIN {X 33.770,Y -29.308,Z -44.953,A -90.000,B 90.000,C 0.000} C_DIS
LIN {X 34.024,Y -29.308,Z -44.935,A -90.000,B 90.000,C 0.000} C_DIS
LIN {X 35.340,Y -29.308,Z -44.887,A -90.000,B 90.000,C 0.000} C_DIS
LIN {X 35.596,Y -29.308,Z -44.900,A -90.000,B 90.000,C 0.000} C_DIS
LIN {X 36.076,Y -29.308,Z -44.928,A -90.000,B 90.000,C 0.000} C_DIS
LIN {X 37.084,Y -29.308,Z -45.005,A -90.000,B 90.000,C 0.000} C_DIS
LIN {X 37.822,Y -29.308,Z -45.052,A -90.000,B 90.000,C 0.000} C_DIS
LIN {X 38.133,Y -29.308,Z -45.069,A -90.000,B 90.000,C 0.000} C_DIS
LIN {X 38.756,Y -29.308,Z -45.050,A -90.000,B 90.000,C 0.000} C_DIS
LIN {X 39.397,Y -29.308,Z -44.912,A -90.000,B 90.000,C 0.000} C_DIS
LIN {X 40.044,Y -29.308,Z -44.703,A -90.000,B 90.000,C 0.000} C_DIS
LIN {X 41.969,Y -29.308,Z -44.073,A -90.000,B 90.000,C 0.000} C_DIS
LIN {X 42.144,Y -29.308,Z -44.012,A -90.000,B 90.000,C 0.000} C_DIS
LIN {X 42.565,Y -29.308,Z -43.882,A -90.000,B 90.000,C 0.000} C_DIS
LIN {X 42.961,Y -29.308,Z -43.787,A -90.000,B 90.000,C 0.000} C_DIS
LIN {X 43.394,Y -29.308,Z -43.705,A -90.000,B 90.000,C 0.000} C_DIS
LIN {X 44.789,Y -29.308,Z -43.454,A -90.000,B 90.000,C 0.000} C_DIS
LIN {X 45.435,Y -29.308,Z -43.402,A -90.000,B 90.000,C 0.000} C_DIS
LIN {X 45.890,Y -29.308,Z -43.393,A -90.000,B 90.000,C 0.000} C_DIS
LIN {X 46.549,Y -29.308,Z -43.387,A -90.000,B 90.000,C 0.000} C_DIS
LIN {X 48.247,Y -29.308,Z -43.541,A -90.000,B 90.000,C 0.000} C_DIS
LIN {X 48.506,Y -29.308,Z -43.582,A -90.000,B 90.000,C 0.000} C_DIS
LIN {X 48.925,Y -29.308,Z -43.666,A -90.000,B 90.000,C 0.000} C_DIS
LIN {X 49.108,Y -29.308,Z -43.710,A -90.000,B 90.000,C 0.000} C_DIS
LIN {X 49.842,Y -29.308,Z -43.904,A -90.000,B 90.000,C 0.000} C_DIS
LIN {X 50.762,Y -29.308,Z -44.204,A -90.000,B 90.000,C 0.000} C_DIS
LIN {X 51.202,Y -29.308,Z -44.360,A -90.000,B 90.000,C 0.000} C_DIS
LIN {X 52.233,Y -29.308,Z -44.761,A -90.000,B 90.000,C 0.000} C_DIS
LIN {X 52.654,Y -29.308,Z -44.963,A -90.000,B 90.000,C 0.000} C_DIS
LIN {X 53.278,Y -29.308,Z -45.282,A -90.000,B 90.000,C 0.000} C_DIS
LIN {X 54.331,Y -29.308,Z -45.858,A -90.000,B 90.000,C 0.000} C_DIS
LIN {X 55.372,Y -29.308,Z -46.441,A -90.000,B 90.000,C 0.000} C_DIS
LIN {X 55.783,Y -29.308,Z -46.708,A -90.000,B 90.000,C 0.000} C_DIS
LIN {X 58.156,Y -29.308,Z -48.571,A -90.000,B 90.000,C 0.000} C_DIS
LIN {X 58.527,Y -29.308,Z -48.870,A -90.000,B 90.000,C 0.000} C_DIS
LIN {X 59.447,Y -29.308,Z -49.710,A -90.000,B 90.000,C 0.000} C_DIS
LIN {X 60.707,Y -29.308,Z -50.848,A -90.000,B 90.000,C 0.000} C_DIS
LIN {X 61.889,Y -29.308,Z -51.975,A -90.000,B 90.000,C 0.000} C_DIS
LIN {X 62.780,Y -29.308,Z -52.820,A -90.000,B 90.000,C 0.000} C_DIS
LIN {X 63.982,Y -29.308,Z -53.904,A -90.000,B 90.000,C 0.000} C_DIS
LIN {X 64.813,Y -29.308,Z -54.661,A -90.000,B 90.000,C 0.000} C_DIS
LIN {X 65.701,Y -29.308,Z -55.365,A -90.000,B 90.000,C 0.000} C_DIS
LIN {X 66.644,Y -29.308,Z -56.091,A -90.000,B 90.000,C 0.000} C_DIS
LIN {X 68.381,Y -29.308,Z -57.385,A -90.000,B 90.000,C 0.000} C_DIS
LIN {X 68.680,Y -29.308,Z -57.599,A -90.000,B 90.000,C 0.000} C_DIS
LIN {X 69.994,Y -29.308,Z -58.598,A -90.000,B 90.000,C 0.000} C_DIS
LIN {X 70.508,Y -29.308,Z -58.989,A -90.000,B 90.000,C 0.000} C_DIS
LIN {X 70.690,Y -29.308,Z -59.122,A -90.000,B 90.000,C 0.000} C_DIS
LIN {X 71.058,Y -29.308,Z -59.409,A -90.000,B 90.000,C 0.000} C_DIS
LIN {X 71.339,Y -29.308,Z -59.649,A -90.000,B 90.000,C 0.000} C_DIS
LIN {X 72.631,Y -29.308,Z -60.796,A -90.000,B 90.000,C 0.000} C_DIS
LIN {X 73.008,Y -29.308,Z -61.145,A -90.000,B 90.000,C 0.000} C_DIS
LIN {X 74.049,Y -29.308,Z -62.331,A -90.000,B 90.000,C 0.000} C_DIS
LIN {X 74.697,Y -29.308,Z -63.083,A -90.000,B 90.000,C 0.000} C_DIS
LIN {X 75.087,Y -29.308,Z -63.620,A -90.000,B 90.000,C 0.000} C_DIS
LIN {X 75.826,Y -29.308,Z -64.617,A -90.000,B 90.000,C 0.000} C_DIS
LIN {X 76.096,Y -29.308,Z -65.011,A -90.000,B 90.000,C 0.000} C_DIS
LIN {X 76.289,Y -29.308,Z -65.317,A -90.000,B 90.000,C 0.000} C_DIS
LIN {X 76.749,Y -29.308,Z -66.054,A -90.000,B 90.000,C 0.000} C_DIS
LIN {X 77.036,Y -29.308,Z -66.470,A -90.000,B 90.000,C 0.000} C_DIS
LIN {X 77.392,Y -29.308,Z -67.055,A -90.000,B 90.000,C 0.000} C_DIS
LIN {X 77.915,Y -29.308,Z -67.827,A -90.000,B 90.000,C 0.000} C_DIS
LIN {X 78.336,Y -29.308,Z -68.439,A -90.000,B 90.000,C 0.000} C_DIS
LIN {X 78.482,Y -29.308,Z -68.658,A -90.000,B 90.000,C 0.000} C_DIS
LIN {X 78.560,Y -29.308,Z -68.762,A -90.000,B 90.000,C 0.000} C_DIS
LIN {X 78.748,Y -29.308,Z -69.023,A -90.000,B 90.000,C 0.000} C_DIS
LIN {X 78.939,Y -29.308,Z -69.288,A -90.000,B 90.000,C 0.000} C_DIS
LIN {X 79.011,Y -29.308,Z -68.759,A -90.000,B 90.000,C 0.000} C_DIS
LIN {X 79.298,Y -29.308,Z -66.972,A -90.000,B 90.000,C 0.000} C_DIS
LIN {X 79.324,Y -29.308,Z -66.863,A -90.000,B 90.000,C 0.000} C_DIS
LIN {X 79.893,Y -29.308,Z -64.655,A -90.000,B 90.000,C 0.000} C_DIS
LIN {X 80.119,Y -29.308,Z -64.023,A -90.000,B 90.000,C 0.000} C_DIS
LIN {X 80.757,Y -29.308,Z -62.329,A -90.000,B 90.000,C 0.000} C_DIS
LIN {X 80.817,Y -29.308,Z -62.172,A -90.000,B 90.000,C 0.000} C_DIS
LIN {X 81.441,Y -29.308,Z -60.611,A -90.000,B 90.000,C 0.000} C_DIS
LIN {X 81.716,Y -29.308,Z -59.971,A -90.000,B 90.000,C 0.000} C_DIS
LIN {X 82.548,Y -29.308,Z -57.960,A -90.000,B 90.000,C 0.000} C_DIS
LIN {X 83.483,Y -29.308,Z -55.948,A -90.000,B 90.000,C 0.000} C_DIS
LIN {X 84.451,Y -29.308,Z -53.781,A -90.000,B 90.000,C 0.000} C_DIS
LIN {X 85.021,Y -29.308,Z -52.625,A -90.000,B 90.000,C 0.000} C_DIS
LIN {X 85.588,Y -29.308,Z -51.550,A -90.000,B 90.000,C 0.000} C_DIS
LIN {X 86.299,Y -29.308,Z -50.356,A -90.000,B 90.000,C 0.000} C_DIS
LIN {X 86.694,Y -29.308,Z -49.736,A -90.000,B 90.000,C 0.000} C_DIS
LIN {X 86.868,Y -29.308,Z -49.476,A -90.000,B 90.000,C 0.000} C_DIS
LIN {X 87.557,Y -29.308,Z -48.511,A -90.000,B 90.000,C 0.000} C_DIS
LIN {X 88.110,Y -29.308,Z -47.786,A -90.000,B 90.000,C 0.000} C_DIS
LIN {X 88.274,Y -29.308,Z -47.579,A -90.000,B 90.000,C 0.000} C_DIS
LIN {X 88.818,Y -29.308,Z -46.941,A -90.000,B 90.000,C 0.000} C_DIS
LIN {X 89.787,Y -29.308,Z -45.868,A -90.000,B 90.000,C 0.000} C_DIS
LIN {X 90.012,Y -29.308,Z -45.641,A -90.000,B 90.000,C 0.000} C_DIS
LIN {X 90.413,Y -29.308,Z -45.243,A -90.000,B 90.000,C 0.000} C_DIS
LIN {X 91.698,Y -29.308,Z -44.051,A -90.000,B 90.000,C 0.000} C_DIS
LIN {X 92.859,Y -29.308,Z -43.126,A -90.000,B 90.000,C 0.000} C_DIS
LIN {X 93.012,Y -29.308,Z -43.010,A -90.000,B 90.000,C 0.000} C_DIS
LIN {X 93.403,Y -29.308,Z -42.720,A -90.000,B 90.000,C 0.000} C_DIS
LIN {X 93.779,Y -29.308,Z -42.446,A -90.000,B 90.000,C 0.000} C_DIS
LIN {X 94.387,Y -29.308,Z -42.041,A -90.000,B 90.000,C 0.000} C_DIS
LIN {X 94.656,Y -29.308,Z -41.864,A -90.000,B 90.000,C 0.000} C_DIS
LIN {X 95.423,Y -29.308,Z -41.379,A -90.000,B 90.000,C 0.000} C_DIS
LIN {X 95.862,Y -29.308,Z -41.122,A -90.000,B 90.000,C 0.000} C_DIS
LIN {X 97.388,Y -29.308,Z -40.253,A -90.000,B 90.000,C 0.000} C_DIS
LIN {X 98.822,Y -29.308,Z -39.515,A -90.000,B 90.000,C 0.000} C_DIS
LIN {X 100.296,Y -29.308,Z -38.817,A -90.000,B 90.000,C 0.000} C_DIS
LIN {X 102.165,Y -29.308,Z -37.970,A -90.000,B 90.000,C 0.000} C_DIS
LIN {X 103.378,Y -29.308,Z -37.428,A -90.000,B 90.000,C 0.000} C_DIS
LIN {X 104.504,Y -29.308,Z -36.930,A -90.000,B 90.000,C 0.000} C_DIS
LIN {X 105.396,Y -29.308,Z -36.555,A -90.000,B 90.000,C 0.000} C_DIS
LIN {X 106.927,Y -29.308,Z -35.947,A -90.000,B 90.000,C 0.000} C_DIS
LIN {X 107.447,Y -29.308,Z -35.751,A -90.000,B 90.000,C 0.000} C_DIS
LIN {X 107.912,Y -29.308,Z -35.585,A -90.000,B 90.000,C 0.000} C_DIS
LIN {X 108.334,Y -29.308,Z -35.444,A -90.000,B 90.000,C 0.000} C_DIS
LIN {X 108.764,Y -29.308,Z -35.329,A -90.000,B 90.000,C 0.000} C_DIS
LIN {X 109.221,Y -29.308,Z -35.225,A -90.000,B 90.000,C 0.000} C_DIS
LIN {X 109.704,Y -29.308,Z -35.162,A -90.000,B 90.000,C 0.000} C_DIS
LIN {X 110.108,Y -29.308,Z -35.113,A -90.000,B 90.000,C 0.000} C_DIS
LIN {X 110.610,Y -29.308,Z -35.105,A -90.000,B 90.000,C 0.000} C_DIS
LIN {X 110.949,Y -29.308,Z -35.117,A -90.000,B 90.000,C 0.000} C_DIS
LIN {X 111.441,Y -29.308,Z -35.159,A -90.000,B 90.000,C 0.000} C_DIS
LIN {X 112.082,Y -29.308,Z -35.281,A -90.000,B 90.000,C 0.000} C_DIS
LIN {X 112.425,Y -29.308,Z -35.368,A -90.000,B 90.000,C 0.000} C_DIS
LIN {X 112.905,Y -29.308,Z -35.512,A -90.000,B 90.000,C 0.000} C_DIS
LIN {X 113.055,Y -29.308,Z -35.560,A -90.000,B 90.000,C 0.000} C_DIS
LIN {X 113.526,Y -29.308,Z -35.756,A -90.000,B 90.000,C 0.000} C_DIS
LIN {X 113.999,Y -29.308,Z -35.983,A -90.000,B 90.000,C 0.000} C_DIS
LIN {X 114.415,Y -29.308,Z -36.208,A -90.000,B 90.000,C 0.000} C_DIS
LIN {X 114.559,Y -29.308,Z -36.298,A -90.000,B 90.000,C 0.000} C_DIS
LIN {X 114.949,Y -29.308,Z -36.564,A -90.000,B 90.000,C 0.000} C_DIS
LIN {X 115.050,Y -29.308,Z -36.644,A -90.000,B 90.000,C 0.000} C_DIS
LIN {X 115.440,Y -29.308,Z -36.974,A -90.000,B 90.000,C 0.000} C_DIS
LIN {X 115.513,Y -29.308,Z -37.039,A -90.000,B 90.000,C 0.000} C_DIS
LIN {X 115.896,Y -29.308,Z -37.436,A -90.000,B 90.000,C 0.000} C_DIS
LIN {X 116.078,Y -29.308,Z -37.630,A -90.000,B 90.000,C 0.000} C_DIS
LIN {X 116.439,Y -29.308,Z -38.088,A -90.000,B 90.000,C 0.000} C_DIS
LIN {X 116.700,Y -29.308,Z -38.500,A -90.000,B 90.000,C 0.000} C_DIS
LIN {X 116.924,Y -29.308,Z -38.953,A -90.000,B 90.000,C 0.000} C_DIS
LIN {X 117.063,Y -29.308,Z -39.259,A -90.000,B 90.000,C 0.000} C_DIS
LIN {X 117.124,Y -29.308,Z -39.417,A -90.000,B 90.000,C 0.000} C_DIS
LIN {X 117.260,Y -29.308,Z -39.781,A -90.000,B 90.000,C 0.000} C_DIS
LIN {X 117.388,Y -29.308,Z -40.270,A -90.000,B 90.000,C 0.000} C_DIS
LIN {X 117.462,Y -29.308,Z -40.593,A -90.000,B 90.000,C 0.000} C_DIS
LIN {X 117.533,Y -29.308,Z -41.051,A -90.000,B 90.000,C 0.000} C_DIS
LIN {X 117.595,Y -29.308,Z -41.513,A -90.000,B 90.000,C 0.000} C_DIS
LIN {X 117.631,Y -29.308,Z -41.898,A -90.000,B 90.000,C 0.000} C_DIS
LIN {X 117.658,Y -29.308,Z -42.426,A -90.000,B 90.000,C 0.000} C_DIS
LIN {X 117.668,Y -29.308,Z -42.692,A -90.000,B 90.000,C 0.000} C_DIS
LIN {X 117.663,Y -29.308,Z -42.910,A -90.000,B 90.000,C 0.000} C_DIS
LIN {X 117.651,Y -29.308,Z -43.202,A -90.000,B 90.000,C 0.000} C_DIS
LIN {X 117.609,Y -29.308,Z -43.709,A -90.000,B 90.000,C 0.000} C_DIS
LIN {X 117.563,Y -29.308,Z -44.141,A -90.000,B 90.000,C 0.000} C_DIS
LIN {X 117.485,Y -29.308,Z -44.657,A -90.000,B 90.000,C 0.000} C_DIS
LIN {X 117.393,Y -29.308,Z -45.143,A -90.000,B 90.000,C 0.000} C_DIS
LIN {X 117.260,Y -29.308,Z -45.739,A -90.000,B 90.000,C 0.000} C_DIS
LIN {X 117.111,Y -29.308,Z -46.241,A -90.000,B 90.000,C 0.000} C_DIS
LIN {X 116.900,Y -29.308,Z -46.938,A -90.000,B 90.000,C 0.000} C_DIS
LIN {X 116.551,Y -29.308,Z -47.845,A -90.000,B 90.000,C 0.000} C_DIS
LIN {X 116.372,Y -29.308,Z -48.278,A -90.000,B 90.000,C 0.000} C_DIS
LIN {X 115.873,Y -29.308,Z -49.350,A -90.000,B 90.000,C 0.000} C_DIS
LIN {X 115.169,Y -29.308,Z -50.757,A -90.000,B 90.000,C 0.000} C_DIS
LIN {X 114.595,Y -29.308,Z -51.893,A -90.000,B 90.000,C 0.000} C_DIS
LIN {X 113.941,Y -29.308,Z -53.229,A -90.000,B 90.000,C 0.000} C_DIS
LIN {X 113.276,Y -29.308,Z -54.687,A -90.000,B 90.000,C 0.000} C_DIS
LIN {X 112.799,Y -29.308,Z -55.830,A -90.000,B 90.000,C 0.000} C_DIS
LIN {X 112.213,Y -29.308,Z -57.388,A -90.000,B 90.000,C 0.000} C_DIS
LIN {X 111.674,Y -29.308,Z -59.009,A -90.000,B 90.000,C 0.000} C_DIS
LIN {X 111.243,Y -29.308,Z -60.507,A -90.000,B 90.000,C 0.000} C_DIS
LIN {X 110.718,Y -29.308,Z -62.430,A -90.000,B 90.000,C 0.000} C_DIS
LIN {X 110.143,Y -29.308,Z -64.468,A -90.000,B 90.000,C 0.000} C_DIS
LIN {X 110.003,Y -29.308,Z -64.938,A -90.000,B 90.000,C 0.000} C_DIS
LIN {X 109.345,Y -29.308,Z -67.050,A -90.000,B 90.000,C 0.000} C_DIS
LIN {X 108.519,Y -29.308,Z -69.358,A -90.000,B 90.000,C 0.000} C_DIS
LIN {X 107.574,Y -29.308,Z -71.736,A -90.000,B 90.000,C 0.000} C_DIS
LIN {X 107.385,Y -29.308,Z -72.191,A -90.000,B 90.000,C 0.000} C_DIS
LIN {X 106.399,Y -29.308,Z -74.452,A -90.000,B 90.000,C 0.000} C_DIS
LIN {X 106.343,Y -29.308,Z -74.568,A -90.000,B 90.000,C 0.000} C_DIS
LIN {X 105.399,Y -29.308,Z -76.539,A -90.000,B 90.000,C 0.000} C_DIS
LIN {X 104.206,Y -29.308,Z -78.767,A -90.000,B 90.000,C 0.000} C_DIS
LIN {X 103.969,Y -29.308,Z -79.179,A -90.000,B 90.000,C 0.000} C_DIS
LIN {X 103.043,Y -29.308,Z -80.750,A -90.000,B 90.000,C 0.000} C_DIS
LIN {X 102.185,Y -29.308,Z -82.097,A -90.000,B 90.000,C 0.000} C_DIS
LIN {X 99.483,Y -29.308,Z -86.142,A -90.000,B 90.000,C 0.000} C_DIS
LIN {X 99.421,Y -29.308,Z -87.027,A -90.000,B 90.000,C 0.000} C_DIS
LIN {X 99.415,Y -29.308,Z -87.635,A -90.000,B 90.000,C 0.000} C_DIS
LIN {X 99.403,Y -29.308,Z -87.958,A -90.000,B 90.000,C 0.000} C_DIS
LIN {X 99.370,Y -29.308,Z -88.704,A -90.000,B 90.000,C 0.000} C_DIS
LIN {X 99.345,Y -29.308,Z -91.048,A -90.000,B 90.000,C 0.000} C_DIS
LIN {X 99.293,Y -29.308,Z -92.402,A -90.000,B 90.000,C 0.000} C_DIS
LIN {X 99.282,Y -29.308,Z -92.642,A -90.000,B 90.000,C 0.000} C_DIS
LIN {X 99.181,Y -29.308,Z -94.099,A -90.000,B 90.000,C 0.000} C_DIS
LIN {X 99.161,Y -29.308,Z -94.258,A -90.000,B 90.000,C 0.000} C_DIS
LIN {X 99.116,Y -29.308,Z -94.573,A -90.000,B 90.000,C 0.000} C_DIS
LIN {X 99.082,Y -29.308,Z -94.782,A -90.000,B 90.000,C 0.000} C_DIS
LIN {X 98.938,Y -29.308,Z -95.534,A -90.000,B 90.000,C 0.000} C_DIS
LIN {X 98.766,Y -29.308,Z -96.309,A -90.000,B 90.000,C 0.000} C_DIS
LIN {X 98.670,Y -29.308,Z -96.727,A -90.000,B 90.000,C 0.000} C_DIS
LIN {X 98.615,Y -29.308,Z -97.027,A -90.000,B 90.000,C 0.000} C_DIS
LIN {X 98.498,Y -29.308,Z -97.489,A -90.000,B 90.000,C 0.000} C_DIS
LIN {X 98.293,Y -29.308,Z -98.191,A -90.000,B 90.000,C 0.000} C_DIS
LIN {X 98.210,Y -29.308,Z -98.611,A -90.000,B 90.000,C 0.000} C_DIS
LIN {X 97.986,Y -29.308,Z -99.869,A -90.000,B 90.000,C 0.000} C_DIS
LIN {X 97.771,Y -29.308,Z -101.168,A -90.000,B 90.000,C 0.000} C_DIS
LIN {X 97.704,Y -29.308,Z -101.623,A -90.000,B 90.000,C 0.000} C_DIS
LIN {X 97.535,Y -29.308,Z -102.917,A -90.000,B 90.000,C 0.000} C_DIS
LIN {X 97.519,Y -29.308,Z -103.028,A -90.000,B 90.000,C 0.000} C_DIS
LIN {X 97.430,Y -29.308,Z -104.057,A -90.000,B 90.000,C 0.000} C_DIS
LIN {X 97.413,Y -29.308,Z -104.213,A -90.000,B 90.000,C 0.000} C_DIS
LIN {X 97.417,Y -29.308,Z -104.998,A -90.000,B 90.000,C 0.000} C_DIS
LIN {X 97.511,Y -29.308,Z -105.860,A -90.000,B 90.000,C 0.000} C_DIS
LIN {X 97.605,Y -29.308,Z -106.424,A -90.000,B 90.000,C 0.000} C_DIS
LIN {X 97.686,Y -29.308,Z -106.929,A -90.000,B 90.000,C 0.000} C_DIS
LIN {X 97.860,Y -29.308,Z -108.137,A -90.000,B 90.000,C 0.000} C_DIS
LIN {X 97.945,Y -29.308,Z -109.257,A -90.000,B 90.000,C 0.000} C_DIS
LIN {X 97.976,Y -29.308,Z -109.626,A -90.000,B 90.000,C 0.000} C_DIS
LIN {X 98.001,Y -29.308,Z -110.081,A -90.000,B 90.000,C 0.000} C_DIS
LIN {X 98.064,Y -29.308,Z -111.553,A -90.000,B 90.000,C 0.000} C_DIS
LIN {X 98.078,Y -29.308,Z -111.812,A -90.000,B 90.000,C 0.000} C_DIS
LIN {X 98.168,Y -29.308,Z -114.962,A -90.000,B 90.000,C 0.000} C_DIS
LIN {X 98.190,Y -29.308,Z -115.828,A -90.000,B 90.000,C 0.000} C_DIS
LIN {X 98.350,Y -29.308,Z -120.359,A -90.000,B 90.000,C 0.000} C_DIS
LIN {X 98.379,Y -29.308,Z -121.454,A -90.000,B 90.000,C 0.000} C_DIS
LIN {X 98.404,Y -29.308,Z -122.553,A -90.000,B 90.000,C 0.000} C_DIS
LIN {X 98.413,Y -29.308,Z -124.845,A -90.000,B 90.000,C 0.000} C_DIS
LIN {X 98.353,Y -29.308,Z -127.212,A -90.000,B 90.000,C 0.000} C_DIS
LIN {X 98.325,Y -29.308,Z -127.722,A -90.000,B 90.000,C 0.000} C_DIS
LIN {X 98.238,Y -29.308,Z -129.475,A -90.000,B 90.000,C 0.000} C_DIS
LIN {X 98.184,Y -29.308,Z -130.236,A -90.000,B 90.000,C 0.000} C_DIS
LIN {X 98.073,Y -29.308,Z -131.918,A -90.000,B 90.000,C 0.000} C_DIS
LIN {X 97.992,Y -29.308,Z -132.961,A -90.000,B 90.000,C 0.000} C_DIS
LIN {X 97.730,Y -29.308,Z -136.519,A -90.000,B 90.000,C 0.000} C_DIS
LIN {X 97.629,Y -29.308,Z -137.844,A -90.000,B 90.000,C 0.000} C_DIS
LIN {X 97.467,Y -29.308,Z -139.854,A -90.000,B 90.000,C 0.000} C_DIS
LIN {X 97.345,Y -29.308,Z -141.326,A -90.000,B 90.000,C 0.000} C_DIS
LIN {X 97.143,Y -29.308,Z -143.481,A -90.000,B 90.000,C 0.000} C_DIS
LIN {X 96.980,Y -29.308,Z -145.160,A -90.000,B 90.000,C 0.000} C_DIS
LIN {X 96.953,Y -29.308,Z -145.421,A -90.000,B 90.000,C 0.000} C_DIS
LIN {X 96.698,Y -29.308,Z -147.683,A -90.000,B 90.000,C 0.000} C_DIS
LIN {X 96.529,Y -29.308,Z -149.123,A -90.000,B 90.000,C 0.000} C_DIS
LIN {X 96.209,Y -29.308,Z -151.409,A -90.000,B 90.000,C 0.000} C_DIS
LIN {X 96.012,Y -29.308,Z -152.744,A -90.000,B 90.000,C 0.000} C_DIS
LIN {X 95.626,Y -29.308,Z -155.058,A -90.000,B 90.000,C 0.000} C_DIS
LIN {X 95.401,Y -29.308,Z -156.322,A -90.000,B 90.000,C 0.000} C_DIS
LIN {X 94.902,Y -29.308,Z -158.895,A -90.000,B 90.000,C 0.000} C_DIS
LIN {X 94.775,Y -29.308,Z -159.534,A -90.000,B 90.000,C 0.000} C_DIS
LIN {X 94.630,Y -29.308,Z -160.235,A -90.000,B 90.000,C 0.000} C_DIS
LIN {X 93.909,Y -29.308,Z -163.547,A -90.000,B 90.000,C 0.000} C_DIS
LIN {X 93.837,Y -29.308,Z -163.854,A -90.000,B 90.000,C 0.000} C_DIS
LIN {X 93.026,Y -29.308,Z -167.232,A -90.000,B 90.000,C 0.000} C_DIS
LIN {X 92.854,Y -29.308,Z -167.899,A -90.000,B 90.000,C 0.000} C_DIS
LIN {X 92.836,Y -29.308,Z -167.976,A -90.000,B 90.000,C 0.000} C_DIS
LIN {X 92.052,Y -29.308,Z -171.034,A -90.000,B 90.000,C 0.000} C_DIS
LIN {X 91.905,Y -29.308,Z -171.654,A -90.000,B 90.000,C 0.000} C_DIS
LIN {X 91.132,Y -29.308,Z -174.548,A -90.000,B 90.000,C 0.000} C_DIS
LIN {X 91.111,Y -29.308,Z -174.635,A -90.000,B 90.000,C 0.000} C_DIS
LIN {X 90.960,Y -29.308,Z -175.262,A -90.000,B 90.000,C 0.000} C_DIS
LIN {X 90.728,Y -29.308,Z -176.138,A -90.000,B 90.000,C 0.000} C_DIS
LIN {X 89.872,Y -29.308,Z -179.297,A -90.000,B 90.000,C 0.000} C_DIS
LIN {X 89.509,Y -29.308,Z -180.870,A -90.000,B 90.000,C 0.000} C_DIS
LIN {X 89.235,Y -29.308,Z -181.912,A -90.000,B 90.000,C 0.000} C_DIS
LIN {X 88.879,Y -29.308,Z -183.559,A -90.000,B 90.000,C 0.000} C_DIS
LIN {X 88.749,Y -29.308,Z -184.078,A -90.000,B 90.000,C 0.000} C_DIS
LIN {X 88.665,Y -29.308,Z -184.503,A -90.000,B 90.000,C 0.000} C_DIS
LIN {X 88.433,Y -29.308,Z -185.727,A -90.000,B 90.000,C 0.000} C_DIS
LIN {X 88.408,Y -29.308,Z -185.926,A -90.000,B 90.000,C 0.000} C_DIS
LIN {X 88.120,Y -29.308,Z -187.671,A -90.000,B 90.000,C 0.000} C_DIS
LIN {X 88.075,Y -29.308,Z -188.131,A -90.000,B 90.000,C 0.000} C_DIS
LIN {X 87.937,Y -29.308,Z -189.748,A -90.000,B 90.000,C 0.000} C_DIS
LIN {X 87.904,Y -29.308,Z -190.066,A -90.000,B 90.000,C 0.000} C_DIS
LIN {X 87.822,Y -29.308,Z -190.703,A -90.000,B 90.000,C 0.000} C_DIS
LIN {X 87.619,Y -29.308,Z -193.138,A -90.000,B 90.000,C 0.000} C_DIS
LIN {X 87.379,Y -29.308,Z -195.508,A -90.000,B 90.000,C 0.000} C_DIS
LIN {X 87.338,Y -29.308,Z -196.087,A -90.000,B 90.000,C 0.000} C_DIS
LIN {X 87.305,Y -29.308,Z -196.404,A -90.000,B 90.000,C 0.000} C_DIS
LIN {X 87.023,Y -29.308,Z -198.459,A -90.000,B 90.000,C 0.000} C_DIS
LIN {X 86.866,Y -29.308,Z -199.842,A -90.000,B 90.000,C 0.000} C_DIS
LIN {X 86.588,Y -29.308,Z -201.417,A -90.000,B 90.000,C 0.000} C_DIS
LIN {X 86.182,Y -29.308,Z -203.946,A -90.000,B 90.000,C 0.000} C_DIS
LIN {X 86.026,Y -29.308,Z -204.724,A -90.000,B 90.000,C 0.000} C_DIS
LIN {X 85.512,Y -29.308,Z -207.491,A -90.000,B 90.000,C 0.000} C_DIS
LIN {X 85.276,Y -29.308,Z -208.590,A -90.000,B 90.000,C 0.000} C_DIS
LIN {X 84.394,Y -29.308,Z -212.429,A -90.000,B 90.000,C 0.000} C_DIS
LIN {X 84.123,Y -29.308,Z -213.630,A -90.000,B 90.000,C 0.000} C_DIS
LIN {X 83.406,Y -29.308,Z -216.665,A -90.000,B 90.000,C 0.000} C_DIS
LIN {X 82.895,Y -29.308,Z -218.923,A -90.000,B 90.000,C 0.000} C_DIS
LIN {X 82.404,Y -29.308,Z -221.006,A -90.000,B 90.000,C 0.000} C_DIS
LIN {X 81.687,Y -29.308,Z -224.307,A -90.000,B 90.000,C 0.000} C_DIS
LIN {X 81.410,Y -29.308,Z -225.409,A -90.000,B 90.000,C 0.000} C_DIS
LIN {X 80.394,Y -29.308,Z -229.845,A -90.000,B 90.000,C 0.000} C_DIS
LIN {X 80.197,Y -29.308,Z -230.586,A -90.000,B 90.000,C 0.000} C_DIS
LIN {X 78.737,Y -29.308,Z -235.877,A -90.000,B 90.000,C 0.000} C_DIS
LIN {X 76.956,Y -29.308,Z -241.169,A -90.000,B 90.000,C 0.000} C_DIS
LIN {X 76.729,Y -29.308,Z -241.872,A -90.000,B 90.000,C 0.000} C_DIS
LIN {X 76.060,Y -29.308,Z -243.561,A -90.000,B 90.000,C 0.000} C_DIS
LIN {X 76.060,Y -60.000,Z -243.561,A -90.000,B 90.000,C 0.000} C_DIS
LIN {X 99.671,Y -60.000,Z -85.862,A -90.000,B 90.000,C 0.000} C_DIS
LIN {X 99.671,Y -27.308,Z -85.862,A -90.000,B 90.000,C 0.000} C_DIS
LIN {X 99.671,Y -27.311,Z -86.034,A -90.000,B 90.000,C 0.000} C_DIS
LIN {X 99.679,Y -27.320,Z -86.230,A -90.000,B 90.000,C 0.000} C_DIS
LIN {X 99.705,Y -27.327,Z -86.861,A -90.000,B 90.000,C 0.000} C_DIS
LIN {X 99.726,Y -27.332,Z -87.318,A -90.000,B 90.000,C 0.000} C_DIS
LIN {X 99.731,Y -27.334,Z -87.646,A -90.000,B 90.000,C 0.000} C_DIS
LIN {X 99.744,Y -27.342,Z -88.522,A -90.000,B 90.000,C 0.000} C_DIS
LIN {X 99.756,Y -27.347,Z -89.286,A -90.000,B 90.000,C 0.000} C_DIS
LIN {X 99.794,Y -27.358,Z -90.505,A -90.000,B 90.000,C 0.000} C_DIS
LIN {X 99.794,Y -27.358,Z -90.575,A -90.000,B 90.000,C 0.000} C_DIS
LIN {X 99.790,Y -27.358,Z -90.850,A -90.000,B 90.000,C 0.000} C_DIS
LIN {X 99.756,Y -27.360,Z -92.134,A -90.000,B 90.000,C 0.000} C_DIS
LIN {X 99.738,Y -27.361,Z -92.673,A -90.000,B 90.000,C 0.000} C_DIS
LIN {X 99.698,Y -27.363,Z -93.385,A -90.000,B 90.000,C 0.000} C_DIS
LIN {X 99.609,Y -27.355,Z -94.137,A -90.000,B 90.000,C 0.000} C_DIS
LIN {X 99.503,Y -27.355,Z -94.863,A -90.000,B 90.000,C 0.000} C_DIS
LIN {X 99.425,Y -27.360,Z -95.390,A -90.000,B 90.000,C 0.000} C_DIS
LIN {X 99.369,Y -27.368,Z -95.825,A -90.000,B 90.000,C 0.000} C_DIS
LIN {X 99.215,Y -27.374,Z -96.632,A -90.000,B 90.000,C 0.000} C_DIS
LIN {X 99.125,Y -27.376,Z -97.101,A -90.000,B 90.000,C 0.000} C_DIS
LIN {X 99.089,Y -27.378,Z -97.290,A -90.000,B 90.000,C 0.000} C_DIS
LIN {X 99.066,Y -27.393,Z -97.588,A -90.000,B 90.000,C 0.000} C_DIS
LIN {X 99.043,Y -27.410,Z -97.871,A -90.000,B 90.000,C 0.000} C_DIS
LIN {X 98.970,Y -27.431,Z -98.330,A -90.000,B 90.000,C 0.000} C_DIS
LIN {X 98.904,Y -27.437,Z -98.735,A -90.000,B 90.000,C 0.000} C_DIS
LIN {X 98.802,Y -27.441,Z -99.374,A -90.000,B 90.000,C 0.000} C_DIS
LIN {X 98.794,Y -27.446,Z -99.487,A -90.000,B 90.000,C 0.000} C_DIS
LIN {X 98.726,Y -27.454,Z -99.992,A -90.000,B 90.000,C 0.000} C_DIS
LIN {X 98.583,Y -27.467,Z -101.048,A -90.000,B 90.000,C 0.000} C_DIS
LIN {X 98.577,Y -27.472,Z -101.149,A -90.000,B 90.000,C 0.000} C_DIS
LIN {X 98.510,Y -27.485,Z -101.798,A -90.000,B 90.000,C 0.000} C_DIS
LIN {X 98.400,Y -27.491,Z -102.739,A -90.000,B 90.000,C 0.000} C_DIS
LIN {X 98.370,Y -27.500,Z -103.109,A -90.000,B 90.000,C 0.000} C_DIS
LIN {X 98.311,Y -27.510,Z -104.017,A -90.000,B 90.000,C 0.000} C_DIS
LIN {X 98.312,Y -27.522,Z -104.258,A -90.000,B 90.000,C 0.000} C_DIS
LIN {X 98.316,Y -27.523,Z -104.431,A -90.000,B 90.000,C 0.000} C_DIS
LIN {X 98.327,Y -27.528,Z -104.801,A -90.000,B 90.000,C 0.000} C_DIS
LIN {X 98.342,Y -27.535,Z -104.955,A -90.000,B 90.000,C 0.000} C_DIS
LIN {X 98.436,Y -27.539,Z -105.733,A -90.000,B 90.000,C 0.000} C_DIS
LIN {X 98.610,Y -27.541,Z -106.780,A -90.000,B 90.000,C 0.000} C_DIS
LIN {X 98.806,Y -27.548,Z -108.072,A -90.000,B 90.000,C 0.000} C_DIS
LIN {X 98.894,Y -27.554,Z -109.074,A -90.000,B 90.000,C 0.000} C_DIS
LIN {X 98.938,Y -27.557,Z -109.541,A -90.000,B 90.000,C 0.000} C_DIS
LIN {X 98.950,Y -27.557,Z -109.748,A -90.000,B 90.000,C 0.000} C_DIS
LIN {X 99.011,Y -27.563,Z -110.853,A -90.000,B 90.000,C 0.000} C_DIS
LIN {X 99.035,Y -27.567,Z -111.236,A -90.000,B 90.000,C 0.000} C_DIS
LIN {X 99.060,Y -27.569,Z -111.691,A -90.000,B 90.000,C 0.000} C_DIS
LIN {X 99.126,Y -27.579,Z -113.331,A -90.000,B 90.000,C 0.000} C_DIS
LIN {X 99.136,Y -27.581,Z -113.540,A -90.000,B 90.000,C 0.000} C_DIS
LIN {X 99.220,Y -27.596,Z -115.697,A -90.000,B 90.000,C 0.000} C_DIS
LIN {X 99.307,Y -27.606,Z -117.726,A -90.000,B 90.000,C 0.000} C_DIS
LIN {X 99.393,Y -27.613,Z -119.823,A -90.000,B 90.000,C 0.000} C_DIS
LIN {X 99.406,Y -27.613,Z -120.179,A -90.000,B 90.000,C 0.000} C_DIS
LIN {X 99.461,Y -27.619,Z -121.953,A -90.000,B 90.000,C 0.000} C_DIS
LIN {X 99.474,Y -27.620,Z -122.466,A -90.000,B 90.000,C 0.000} C_DIS
LIN {X 99.501,Y -27.630,Z -124.821,A -90.000,B 90.000,C 0.000} C_DIS
LIN {X 99.455,Y -27.640,Z -127.240,A -90.000,B 90.000,C 0.000} C_DIS
LIN {X 99.429,Y -27.641,Z -127.771,A -90.000,B 90.000,C 0.000} C_DIS
LIN {X 99.353,Y -27.649,Z -129.531,A -90.000,B 90.000,C 0.000} C_DIS
LIN {X 99.315,Y -27.652,Z -130.122,A -90.000,B 90.000,C 0.000} C_DIS
LIN {X 99.200,Y -27.658,Z -132.005,A -90.000,B 90.000,C 0.000} C_DIS
LIN {X 99.140,Y -27.661,Z -132.815,A -90.000,B 90.000,C 0.000} C_DIS
LIN {X 98.999,Y -27.666,Z -134.832,A -90.000,B 90.000,C 0.000} C_DIS
LIN {X 98.872,Y -27.669,Z -136.606,A -90.000,B 90.000,C 0.000} C_DIS
LIN {X 98.773,Y -27.671,Z -137.936,A -90.000,B 90.000,C 0.000} C_DIS
LIN {X 98.615,Y -27.673,Z -139.949,A -90.000,B 90.000,C 0.000} C_DIS
LIN {X 98.494,Y -27.675,Z -141.433,A -90.000,B 90.000,C 0.000} C_DIS
LIN {X 98.297,Y -27.679,Z -143.593,A -90.000,B 90.000,C 0.000} C_DIS
LIN {X 98.155,Y -27.681,Z -145.103,A -90.000,B 90.000,C 0.000} C_DIS
LIN {X 98.108,Y -27.681,Z -145.551,A -90.000,B 90.000,C 0.000} C_DIS
LIN {X 97.862,Y -27.688,Z -147.819,A -90.000,B 90.000,C 0.000} C_DIS
LIN {X 97.700,Y -27.691,Z -149.239,A -90.000,B 90.000,C 0.000} C_DIS
LIN {X 97.359,Y -27.704,Z -151.800,A -90.000,B 90.000,C 0.000} C_DIS
LIN {X 97.207,Y -27.708,Z -152.860,A -90.000,B 90.000,C 0.000} C_DIS
LIN {X 97.157,Y -27.709,Z -153.181,A -90.000,B 90.000,C 0.000} C_DIS
LIN {X 96.979,Y -27.717,Z -154.311,A -90.000,B 90.000,C 0.000} C_DIS
LIN {X 96.790,Y -27.727,Z -155.498,A -90.000,B 90.000,C 0.000} C_DIS
LIN {X 96.627,Y -27.732,Z -156.450,A -90.000,B 90.000,C 0.000} C_DIS
LIN {X 96.180,Y -27.753,Z -158.912,A -90.000,B 90.000,C 0.000} C_DIS
LIN {X 95.963,Y -27.768,Z -160.092,A -90.000,B 90.000,C 0.000} C_DIS
LIN {X 95.881,Y -27.771,Z -160.508,A -90.000,B 90.000,C 0.000} C_DIS
LIN {X 95.776,Y -27.778,Z -161.023,A -90.000,B 90.000,C 0.000} C_DIS
LIN {X 95.203,Y -27.809,Z -163.826,A -90.000,B 90.000,C 0.000} C_DIS
LIN {X 94.963,Y -27.839,Z -164.970,A -90.000,B 90.000,C 0.000} C_DIS
LIN {X 94.383,Y -27.870,Z -167.532,A -90.000,B 90.000,C 0.000} C_DIS
LIN {X 94.138,Y -27.901,Z -168.618,A -90.000,B 90.000,C 0.000} C_DIS
LIN {X 93.505,Y -27.936,Z -171.225,A -90.000,B 90.000,C 0.000} C_DIS
LIN {X 93.473,Y -27.940,Z -171.363,A -90.000,B 90.000,C 0.000} C_DIS
LIN {X 93.334,Y -27.951,Z -171.993,A -90.000,B 90.000,C 0.000} C_DIS
LIN {X 93.049,Y -27.984,Z -173.179,A -90.000,B 90.000,C 0.000} C_DIS
LIN {X 92.643,Y -28.008,Z -174.781,A -90.000,B 90.000,C 0.000} C_DIS
LIN {X 92.614,Y -28.012,Z -174.900,A -90.000,B 90.000,C 0.000} C_DIS
LIN {X 92.569,Y -28.016,Z -175.101,A -90.000,B 90.000,C 0.000} C_DIS
LIN {X 92.461,Y -28.025,Z -175.584,A -90.000,B 90.000,C 0.000} C_DIS
LIN {X 92.218,Y -28.057,Z -176.604,A -90.000,B 90.000,C 0.000} C_DIS
LIN {X 91.931,Y -28.076,Z -177.721,A -90.000,B 90.000,C 0.000} C_DIS
LIN {X 91.587,Y -28.101,Z -179.066,A -90.000,B 90.000,C 0.000} C_DIS
LIN {X 91.443,Y -28.125,Z -179.663,A -90.000,B 90.000,C 0.000} C_DIS
LIN {X 91.189,Y -28.152,Z -180.853,A -90.000,B 90.000,C 0.000} C_DIS
LIN {X 91.151,Y -28.154,Z -181.022,A -90.000,B 90.000,C 0.000} C_DIS
LIN {X 91.110,Y -28.157,Z -181.209,A -90.000,B 90.000,C 0.000} C_DIS
LIN {X 90.858,Y -28.206,Z -182.301,A -90.000,B 90.000,C 0.000} C_DIS
LIN {X 90.600,Y -28.238,Z -183.596,A -90.000,B 90.000,C 0.000} C_DIS
LIN {X 90.539,Y -28.250,Z -183.909,A -90.000,B 90.000,C 0.000} C_DIS
LIN {X 90.419,Y -28.277,Z -184.465,A -90.000,B 90.000,C 0.000} C_DIS
LIN {X 90.270,Y -28.301,Z -185.312,A -90.000,B 90.000,C 0.000} C_DIS
LIN {X 90.214,Y -28.316,Z -185.657,A -90.000,B 90.000,C 0.000} C_DIS
LIN {X 90.156,Y -28.329,Z -186.002,A -90.000,B 90.000,C 0.000} C_DIS
LIN {X 90.142,Y -28.331,Z -186.117,A -90.000,B 90.000,C 0.000} C_DIS
LIN {X 89.997,Y -28.357,Z -187.097,A -90.000,B 90.000,C 0.000} C_DIS
LIN {X 89.883,Y -28.393,Z -187.904,A -90.000,B 90.000,C 0.000} C_DIS
LIN {X 89.855,Y -28.398,Z -188.219,A -90.000,B 90.000,C 0.000} C_DIS
LIN {X 89.775,Y -28.402,Z -189.180,A -90.000,B 90.000,C 0.000} C_DIS
LIN {X 89.721,Y -28.417,Z -189.901,A -90.000,B 90.000,C 0.000} C_DIS
LIN {X 89.691,Y -28.427,Z -190.237,A -90.000,B 90.000,C 0.000} C_DIS
LIN {X 89.655,Y -28.439,Z -190.566,A -90.000,B 90.000,C 0.000} C_DIS
LIN {X 89.621,Y -28.445,Z -190.850,A -90.000,B 90.000,C 0.000} C_DIS
LIN {X 89.585,Y -28.446,Z -191.280,A -90.000,B 90.000,C 0.000} C_DIS
LIN {X 89.442,Y -28.478,Z -193.178,A -90.000,B 90.000,C 0.000} C_DIS
LIN {X 89.424,Y -28.478,Z -193.374,A -90.000,B 90.000,C 0.000} C_DIS
LIN {X 89.290,Y -28.492,Z -194.757,A -90.000,B 90.000,C 0.000} C_DIS
LIN {X 89.202,Y -28.493,Z -195.635,A -90.000,B 90.000,C 0.000} C_DIS
LIN {X 89.164,Y -28.489,Z -196.122,A -90.000,B 90.000,C 0.000} C_DIS
LIN {X 89.157,Y -28.487,Z -196.214,A -90.000,B 90.000,C 0.000} C_DIS
LIN {X 89.138,Y -28.487,Z -196.405,A -90.000,B 90.000,C 0.000} C_DIS
LIN {X 89.118,Y -28.484,Z -196.593,A -90.000,B 90.000,C 0.000} C_DIS
LIN {X 88.829,Y -28.479,Z -198.685,A -90.000,B 90.000,C 0.000} C_DIS
LIN {X 88.686,Y -28.466,Z -199.886,A -90.000,B 90.000,C 0.000} C_DIS
LIN {X 88.666,Y -28.461,Z -200.047,A -90.000,B 90.000,C 0.000} C_DIS
LIN {X 88.649,Y -28.459,Z -200.156,A -90.000,B 90.000,C 0.000} C_DIS
LIN {X 88.375,Y -28.451,Z -201.689,A -90.000,B 90.000,C 0.000} C_DIS
LIN {X 87.986,Y -28.424,Z -204.028,A -90.000,B 90.000,C 0.000} C_DIS
LIN {X 87.951,Y -28.419,Z -204.230,A -90.000,B 90.000,C 0.000} C_DIS
LIN {X 87.785,Y -28.414,Z -205.050,A -90.000,B 90.000,C 0.000} C_DIS
LIN {X 87.245,Y -28.382,Z -207.863,A -90.000,B 90.000,C 0.000} C_DIS
LIN {X 87.008,Y -28.380,Z -208.962,A -90.000,B 90.000,C 0.000} C_DIS
LIN {X 86.902,Y -28.381,Z -209.425,A -90.000,B 90.000,C 0.000} C_DIS
LIN {X 86.125,Y -28.384,Z -212.819,A -90.000,B 90.000,C 0.000} C_DIS
LIN {X 85.852,Y -28.382,Z -214.021,A -90.000,B 90.000,C 0.000} C_DIS
LIN {X 85.243,Y -28.386,Z -216.609,A -90.000,B 90.000,C 0.000} C_DIS
LIN {X 85.167,Y -28.385,Z -216.929,A -90.000,B 90.000,C 0.000} C_DIS
LIN {X 84.608,Y -28.359,Z -219.327,A -90.000,B 90.000,C 0.000} C_DIS
LIN {X 84.116,Y -28.349,Z -221.394,A -90.000,B 90.000,C 0.000} C_DIS
LIN {X 83.660,Y -28.322,Z -223.421,A -90.000,B 90.000,C 0.000} C_DIS
LIN {X 83.381,Y -28.310,Z -224.675,A -90.000,B 90.000,C 0.000} C_DIS
LIN {X 83.357,Y -28.311,Z -224.773,A -90.000,B 90.000,C 0.000} C_DIS
LIN {X 83.098,Y -28.308,Z -225.795,A -90.000,B 90.000,C 0.000} C_DIS
LIN {X 82.581,Y -28.278,Z -227.972,A -90.000,B 90.000,C 0.000} C_DIS
LIN {X 82.056,Y -28.260,Z -230.220,A -90.000,B 90.000,C 0.000} C_DIS
LIN {X 81.994,Y -28.262,Z -230.460,A -90.000,B 90.000,C 0.000} C_DIS
LIN {X 81.841,Y -28.256,Z -231.023,A -90.000,B 90.000,C 0.000} C_DIS
LIN {X 81.370,Y -28.245,Z -232.703,A -90.000,B 90.000,C 0.000} C_DIS
LIN {X 80.409,Y -28.246,Z -236.187,A -90.000,B 90.000,C 0.000} C_DIS
LIN {X 80.369,Y -28.242,Z -236.327,A -90.000,B 90.000,C 0.000} C_DIS
LIN {X 80.340,Y -28.241,Z -236.417,A -90.000,B 90.000,C 0.000} C_DIS
LIN {X 79.887,Y -28.241,Z -237.763,A -90.000,B 90.000,C 0.000} C_DIS
LIN {X 78.580,Y -28.265,Z -241.691,A -90.000,B 90.000,C 0.000} C_DIS
LIN {X 78.411,Y -28.265,Z -242.218,A -90.000,B 90.000,C 0.000} C_DIS
LIN {X 78.350,Y -28.260,Z -242.395,A -90.000,B 90.000,C 0.000} C_DIS
LIN {X 78.312,Y -28.258,Z -242.499,A -90.000,B 90.000,C 0.000} C_DIS
LIN {X 78.018,Y -28.258,Z -243.240,A -90.000,B 90.000,C 0.000} C_DIS
LIN {X 77.892,Y -28.260,Z -243.561,A -90.000,B 90.000,C 0.000} C_DIS
LIN {X 77.892,Y -60.000,Z -243.561,A -90.000,B 90.000,C 0.000} C_DIS
LIN {X 92.237,Y -60.000,Z -184.394,A -90.000,B 90.000,C 0.000} C_DIS
LIN {X 92.237,Y -27.308,Z -184.394,A -90.000,B 90.000,C 0.000} C_DIS
LIN {X 92.145,Y -27.338,Z -184.841,A -90.000,B 90.000,C 0.000} C_DIS
